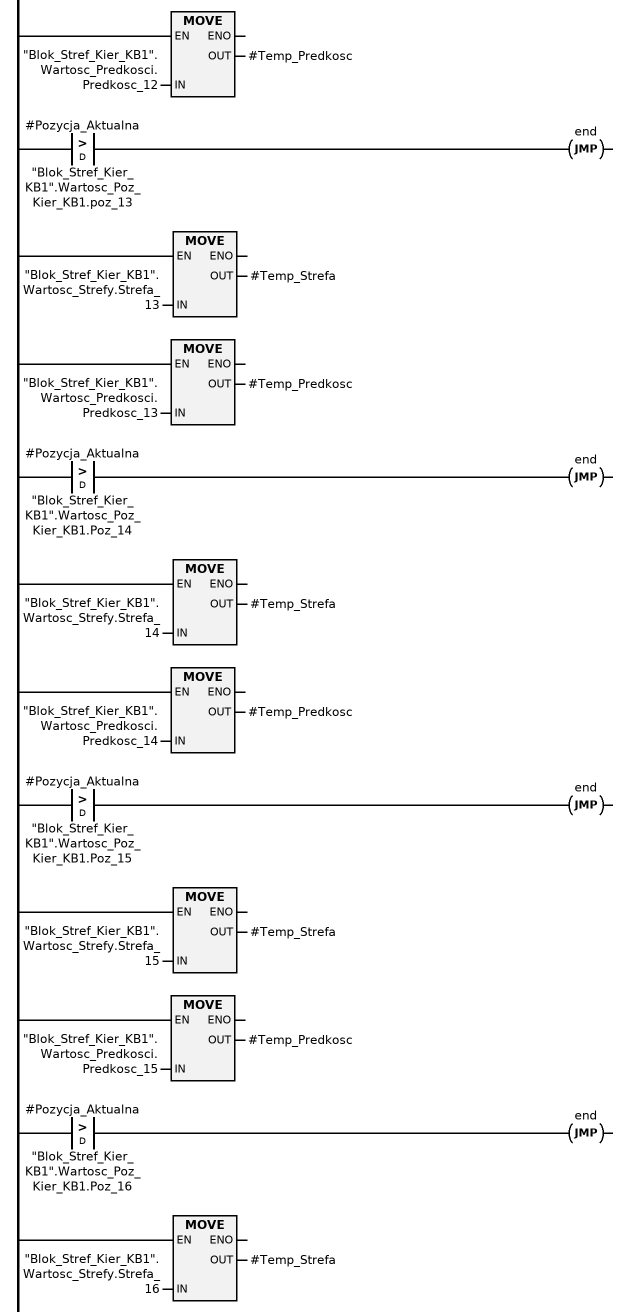
[picture p382: Przelaczanie_Stref_K_KB1 networks 3-3]
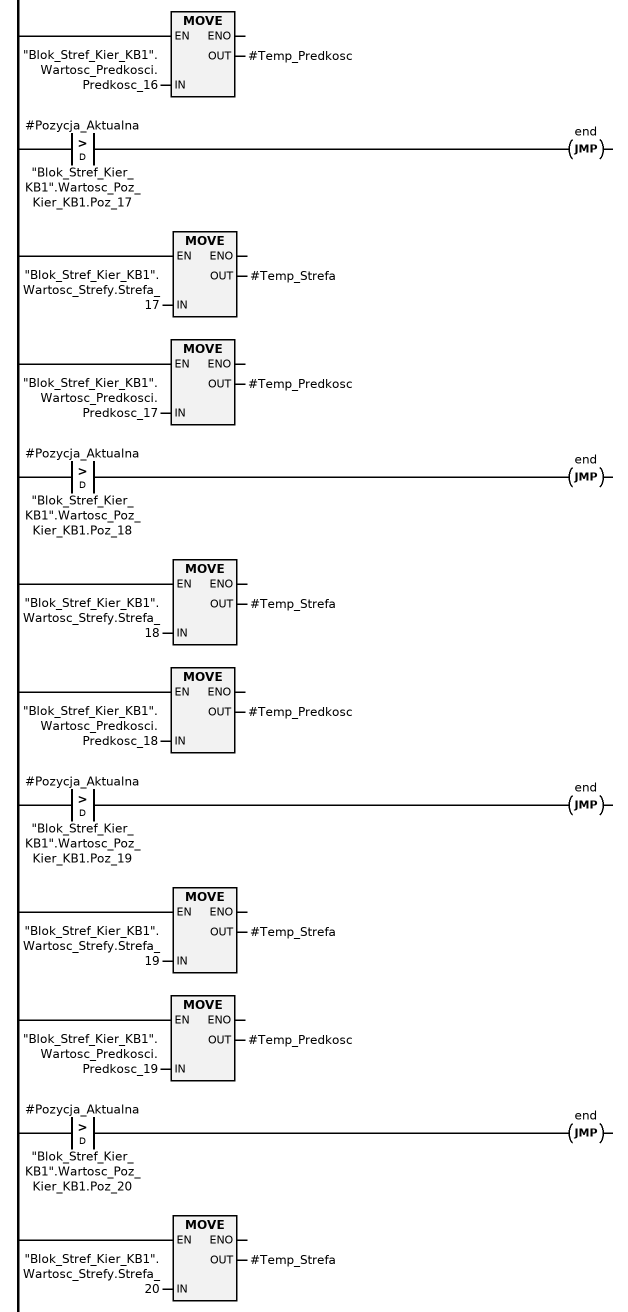
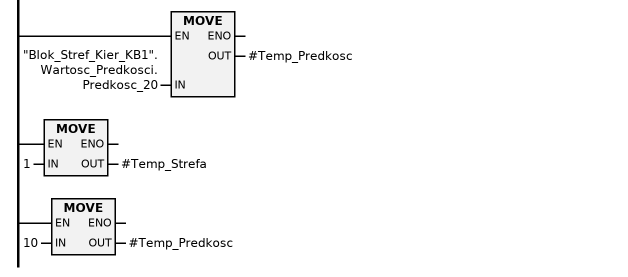
NETWORK
TITLE =
//Porowanie Pozycji z zadana strefa
//
//B1       
//
//5000               
//
//10000
//
//KB2
//                        /\
//                        |
//12000                 Wozek
//
//
//Gender
//15000
//*********Poz  0
      L     #Pozycja_Aktualna;	//np 350000
      L     "Blok_Stref_Kier_KB1".Wartosc_Poz_Kier_KB1.Poz_0;	//np40000 idzie dalej
      >D;
      JC    end;
      L     "Blok_Stref_Kier_KB1".Wartosc_Strefy.Strefa_0;
      T     #Temp_Strefa;
      L     "Blok_Stref_Kier_KB1".Wartosc_Predkosci.Predkosc_0;
      T     #Temp_Predkosc;
//*********Poz  1
      L     #Pozycja_Aktualna;	//30000
      L     "Blok_Stref_Kier_KB1".Wartosc_Poz_Kier_KB1.Poz_1;	//np.24000 tu zostaje
      >D;
      JC    end;
      L     "Blok_Stref_Kier_KB1".Wartosc_Strefy.Strefa_1;
      T     #Temp_Strefa;
      L     "Blok_Stref_Kier_KB1".Wartosc_Predkosci.Predkosc_1;
      T     #Temp_Predkosc;
//********Poz 2
      L     #Pozycja_Aktualna;	//20000
      L     "Blok_Stref_Kier_KB1".Wartosc_Poz_Kier_KB1.Poz_2;	//np22000
      >D;
      JC    end;
      L     "Blok_Stref_Kier_KB1".Wartosc_Strefy.Strefa_2;
      T     #Temp_Strefa;
      L     "Blok_Stref_Kier_KB1".Wartosc_Predkosci.Predkosc_2;
      T     #Temp_Predkosc;
//********Poz 3
      L     #Pozycja_Aktualna;
      L     "Blok_Stref_Kier_KB1".Wartosc_Poz_Kier_KB1.Poz_3;
      >D;
      JC    end;
      L     "Blok_Stref_Kier_KB1".Wartosc_Strefy.Strefa_3;
      T     #Temp_Strefa;
      L     "Blok_Stref_Kier_KB1".Wartosc_Predkosci.Predkosc_3;
      T     #Temp_Predkosc;
//********Poz 4
      L     #Pozycja_Aktualna;
      L     "Blok_Stref_Kier_KB1".Wartosc_Poz_Kier_KB1.Poz_4;
      >D;
      JC    end;
      L     "Blok_Stref_Kier_KB1".Wartosc_Strefy.Strefa_4;
      T     #Temp_Strefa;
      L     "Blok_Stref_Kier_KB1".Wartosc_Predkosci.Predkosc_4;
      T     #Temp_Predkosc;
//********Poz 5
      L     #Pozycja_Aktualna;
      L     "Blok_Stref_Kier_KB1".Wartosc_Poz_Kier_KB1.Poz_5;
      >D;
      JC    end;
      L     "Blok_Stref_Kier_KB1".Wartosc_Strefy.Strefa_5;
      T     #Temp_Strefa;
      L     "Blok_Stref_Kier_KB1".Wartosc_Predkosci.Predkosc_5;
      T     #Temp_Predkosc;
//********Poz 6
      L     #Pozycja_Aktualna;
      L     "Blok_Stref_Kier_KB1".Wartosc_Poz_Kier_KB1.Poz_6;
      >D;
      JC    end;
      L     "Blok_Stref_Kier_KB1".Wartosc_Strefy.Strefa_6;
      T     #Temp_Strefa;
      L     "Blok_Stref_Kier_KB1".Wartosc_Predkosci.Predkosc_6;
      T     #Temp_Predkosc;
//********Poz 7
      L     #Pozycja_Aktualna;
      L     "Blok_Stref_Kier_KB1".Wartosc_Poz_Kier_KB1.Poz_7;
      >D;
      JC    end;
      L     "Blok_Stref_Kier_KB1".Wartosc_Strefy.Strefa_7;
      T     #Temp_Strefa;
      L     "Blok_Stref_Kier_KB1".Wartosc_Predkosci.Predkosc_7;
      T     #Temp_Predkosc;
//********Poz 8
      L     #Pozycja_Aktualna;
      L     "Blok_Stref_Kier_KB1".Wartosc_Poz_Kier_KB1.Poz_8;
      >D;
      JC    end;
      L     "Blok_Stref_Kier_KB1".Wartosc_Strefy.Strefa_8;
      T     #Temp_Strefa;
      L     "Blok_Stref_Kier_KB1".Wartosc_Predkosci.Predkosc_8;
      T     #Temp_Predkosc;
//********Poz 9
      L     #Pozycja_Aktualna;
      L     "Blok_Stref_Kier_KB1".Wartosc_Poz_Kier_KB1.Poz_9;
      >D;
      JC    end;
      L     "Blok_Stref_Kier_KB1".Wartosc_Strefy.Strefa_9;
      T     #Temp_Strefa;
      L     "Blok_Stref_Kier_KB1".Wartosc_Predkosci.Predkosc_9;
      T     #Temp_Predkosc;
//********Poz 10
      L     #Pozycja_Aktualna;
      L     "Blok_Stref_Kier_KB1".Wartosc_Poz_Kier_KB1.Poz_10;
      >D;
      JC    end;
      L     "Blok_Stref_Kier_KB1".Wartosc_Strefy.Strefa_10;
      T     #Temp_Strefa;
      L     "Blok_Stref_Kier_KB1".Wartosc_Predkosci.Predkosc_10;
      T     #Temp_Predkosc;
//********Poz 11
      L     #Pozycja_Aktualna;
      L     "Blok_Stref_Kier_KB1".Wartosc_Poz_Kier_KB1.Poz_11;
      >D;
      JC    end;
      L     "Blok_Stref_Kier_KB1".Wartosc_Strefy.Strefa_11;
      T     #Temp_Strefa;
      L     "Blok_Stref_Kier_KB1".Wartosc_Predkosci.Predkosc_11;
      T     #Temp_Predkosc;
//********Poz 12
      L     #Pozycja_Aktualna;
      L     "Blok_Stref_Kier_KB1".Wartosc_Poz_Kier_KB1.Poz_12;
      >D;
      JC    end;
      L     "Blok_Stref_Kier_KB1".Wartosc_Strefy.Strefa_12;
      T     #Temp_Strefa;
      L     "Blok_Stref_Kier_KB1".Wartosc_Predkosci.Predkosc_12;
      T     #Temp_Predkosc;
//********Poz 13
      L     #Pozycja_Aktualna;
      L     "Blok_Stref_Kier_KB1".Wartosc_Poz_Kier_KB1.poz_13;
      >D;
      JC    end;
      L     "Blok_Stref_Kier_KB1".Wartosc_Strefy.Strefa_13;
      T     #Temp_Strefa;
      L     "Blok_Stref_Kier_KB1".Wartosc_Predkosci.Predkosc_13;
      T     #Temp_Predkosc;
//********Poz 14
      L     #Pozycja_Aktualna;
      L     "Blok_Stref_Kier_KB1".Wartosc_Poz_Kier_KB1.Poz_14;
      >D;
      JC    end;
      L     "Blok_Stref_Kier_KB1".Wartosc_Strefy.Strefa_14;
      T     #Temp_Strefa;
      L     "Blok_Stref_Kier_KB1".Wartosc_Predkosci.Predkosc_14;
      T     #Temp_Predkosc;
//********Poz 15
      L     #Pozycja_Aktualna;
      L     "Blok_Stref_Kier_KB1".Wartosc_Poz_Kier_KB1.Poz_15;
      >D;
      JC    end;
      L     "Blok_Stref_Kier_KB1".Wartosc_Strefy.Strefa_15;
      T     #Temp_Strefa;
      L     "Blok_Stref_Kier_KB1".Wartosc_Predkosci.Predkosc_15;
      T     #Temp_Predkosc;
//********Poz 16
      L     #Pozycja_Aktualna;
      L     "Blok_Stref_Kier_KB1".Wartosc_Poz_Kier_KB1.Poz_16;
      >D;
      JC    end;
      L     "Blok_Stref_Kier_KB1".Wartosc_Strefy.Strefa_16;
      T     #Temp_Strefa;
      L     "Blok_Stref_Kier_KB1".Wartosc_Predkosci.Predkosc_16;
      T     #Temp_Predkosc;
//********Poz 17
      L     #Pozycja_Aktualna;
      L     "Blok_Stref_Kier_KB1".Wartosc_Poz_Kier_KB1.Poz_17;
      >D;
      JC    end;
      L     "Blok_Stref_Kier_KB1".Wartosc_Strefy.Strefa_17;
      T     #Temp_Strefa;
      L     "Blok_Stref_Kier_KB1".Wartosc_Predkosci.Predkosc_17;
      T     #Temp_Predkosc;
//********Poz 18
      L     #Pozycja_Aktualna;
      L     "Blok_Stref_Kier_KB1".Wartosc_Poz_Kier_KB1.Poz_18;
      >D;
      JC    end;
      L     "Blok_Stref_Kier_KB1".Wartosc_Strefy.Strefa_18;
      T     #Temp_Strefa;
      L     "Blok_Stref_Kier_KB1".Wartosc_Predkosci.Predkosc_18;
      T     #Temp_Predkosc;
//********Poz 19
      L     #Pozycja_Aktualna;
      L     "Blok_Stref_Kier_KB1".Wartosc_Poz_Kier_KB1.Poz_19;
      >D;
      JC    end;
      L     "Blok_Stref_Kier_KB1".Wartosc_Strefy.Strefa_19;
      T     #Temp_Strefa;
      L     "Blok_Stref_Kier_KB1".Wartosc_Predkosci.Predkosc_19;
      T     #Temp_Predkosc;
//********Poz 20
      L     #Pozycja_Aktualna;
      L     "Blok_Stref_Kier_KB1".Wartosc_Poz_Kier_KB1.Poz_20;
      >D;
      JC    end;
      L     "Blok_Stref_Kier_KB1".Wartosc_Strefy.Strefa_20;
      T     #Temp_Strefa;
      L     "Blok_Stref_Kier_KB1".Wartosc_Predkosci.Predkosc_20;
      T     #Temp_Predkosc;
//Jezeli nic nie wyszlo wybierz strefe najwieksza
      L     1;
      T     #Temp_Strefa;
      L     10;
      T     #Temp_Predkosc;
end:  NOP   0;
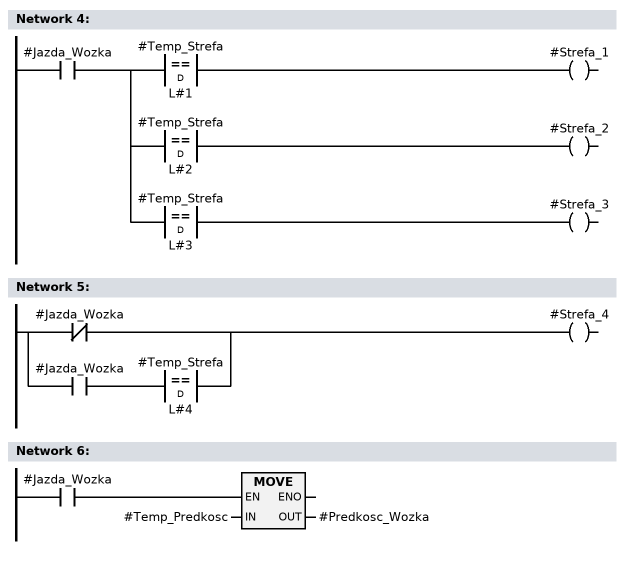
NETWORK
TITLE =
//Przypisanie predkosc. Strefa 1 to strefa podluzna.
//
      A     #Jazda_Wozka;
      =     L 8.0;
      A     L 8.0;
      A(;
      L     #Temp_Strefa;
      L     L#1;
      ==D;
      );
      =     #Strefa_1;
      A     L 8.0;
      A(;
      L     #Temp_Strefa;
      L     L#2;
      ==D;
      );
      =     #Strefa_2;
      A     L 8.0;
      A(;
      L     #Temp_Strefa;
      L     L#3;
      ==D;
      );
      =     #Strefa_3;
NETWORK
TITLE =
//Jezeli wozek stoi
      ON    #Jazda_Wozka;
      O;
      A     #Jazda_Wozka;
      A(;
      L     #Temp_Strefa;
      L     L#4;
      ==D;
      );
      =     #Strefa_4;
NETWORK
TITLE =
//Przyporzadkowanie predkosci
      A     #Jazda_Wozka;
      JNB   _001;
      L     #Temp_Predkosc;
      T     #Predkosc_Wozka;
_001: NOP   0;
END_FUNCTION

FUNCTION "Blok_Bedow" : VOID	// FC 119
//Funkcja obslugujaca bledy
VERSION : 0.1
BEGIN
NETWORK
TITLE =
//Ten network celowo jest wolny
//
NETWORK
TITLE =
END_FUNCTION

FUNCTION "Fal_Sew" : VOID	// FC 140
//Dieses Programmbeispiel zeigt nur die prinzipielle Vorgehensweise.
//Für fehlerhafte Programmfunktionen und deren Folgen
//kann weder eine juristische, noch irgendeine Haftung übernommen werden!
//
//Eingänge der FC:
//"DRIVE_IO_ADDRESS": Anfangsadresse des E/A-Bereichs => Hardwarekonfiguration
//"ENABLE_RAPID_STOP" = true: Freigabe; false: Schnellstopp
//"RESET": Fehler quittieren
//Die Betriebsart wird mit den Eingängen "Jog_plus_mode, Jog_minus_mode; 
//Ref_travel und Positioning_mode angewählt.
//"SETPOINT_POS": Positionssollwert (DINT) in Anwendereinheit.
//Die Anwendereinheit ist abhängig von der Inbetriebnahme der "Erweiterten 
//Buspositionierung"
//"SETPOINT_SPEED": Positioniergeschwindigkeit (INT) in rpm
//"START_RAMP": Beschleunigungsrampe (INT) in ms
//"STOP_RAMP": Verzögerungsrampe(INT) in ms
AUTHOR : SG-MEST
FAMILY : PROFIBUS
NAME : MDX_POS
VERSION : 1.1
VAR_INPUT
  DRIVE_IO_ADDRESS : INT ;
  ENABLE_RAPID_STOP : BOOL ;
  RESET : BOOL ;
  JOG_PLUS_MODE : BOOL ;
  JOG_MINUS_MODE : BOOL ;
  REF_TRAVEL_MODE : BOOL ;
  POSITIONING_MODE : BOOL ;
  SETPOINT_POS : DINT ;	//in mm
  SETPOINT_SPEED : INT ;	//Positioniergeschwindigkeit (INT) in rpm (1350rpm)
  START_RAMP : INT ;	//Beschleunigungsrampe (INT) in ms
  STOP_RAMP : INT ;	//Verzögerungsrampe(INT) in ms
END_VAR
VAR_OUTPUT
  COMMUNICATION_OK : BOOL ;	//SFC14/SFC15: Return Value = 0
  FAULT_OF_AXIS : BOOL ;
  WARNING_OF_AXIS : BOOL ;
  INVERTER_READY : BOOL ;
  REFERENCED : BOOL ;
  TARGET_POS_REACHED : BOOL ;
  AXIS_INTERLOCKED : BOOL ;	//die Modeanwahl ist unplausibel (kein Mode oder mehrere Modi angewählt)
  FAULT_NO : INT ;
  ACTUAL_POSITION : DINT ;
  ACTUAL_SPEED : INT ;
  ACTUAL_CURRENT : INT ;
END_VAR
VAR_TEMP
  PI : STRUCT
   Status : BYTE ;
   Motor_turning : BOOL ;
   Inverter_ready : BOOL ;
   referenced : BOOL ;
   Target_position_reached : BOOL ;
   Brake_released : BOOL ;
   Error : BOOL ;
   Limit_Switch_CW : BOOL ;
   Limit_switch_CCW : BOOL ;
   Actual_position : DINT ;
   Actual_speed : INT ;
   Active_current : INT ;
   Device_utilisation : INT ;
  END_STRUCT ;
  PO : STRUCT
   start : BOOL ;
   Jog_plus : BOOL ;
   Jog_minus : BOOL ;
   mode_low : BOOL ;
   mode_high : BOOL ;
   CTW_Bit_13 : BOOL ;
   CTW_Bit_14 : BOOL ;
   CTW_Bit_15 : BOOL ;
   Contr_inhibit : BOOL ;
   Rapid_stop : BOOL ;
   Stop : BOOL ;
   CTW_Bit_3 : BOOL ;
   CTW_Bit_4 : BOOL ;
   CTW_Bit_5 : BOOL ;
   Reset_fault : BOOL ;
   CTW_Bit_7 : BOOL ;
   Setpoint_position : DINT ;
   Setpoint_speed : INT ;
   Start_ramp : INT ;
   Stop_ramp : INT ;
  END_STRUCT ;
  Ref : BOOL ;
  Pos : BOOL ;
  Addr : WORD ;
  Returncode_SFC14 : INT ;
  Returncode_SFC15 : INT ;
END_VAR
BEGIN
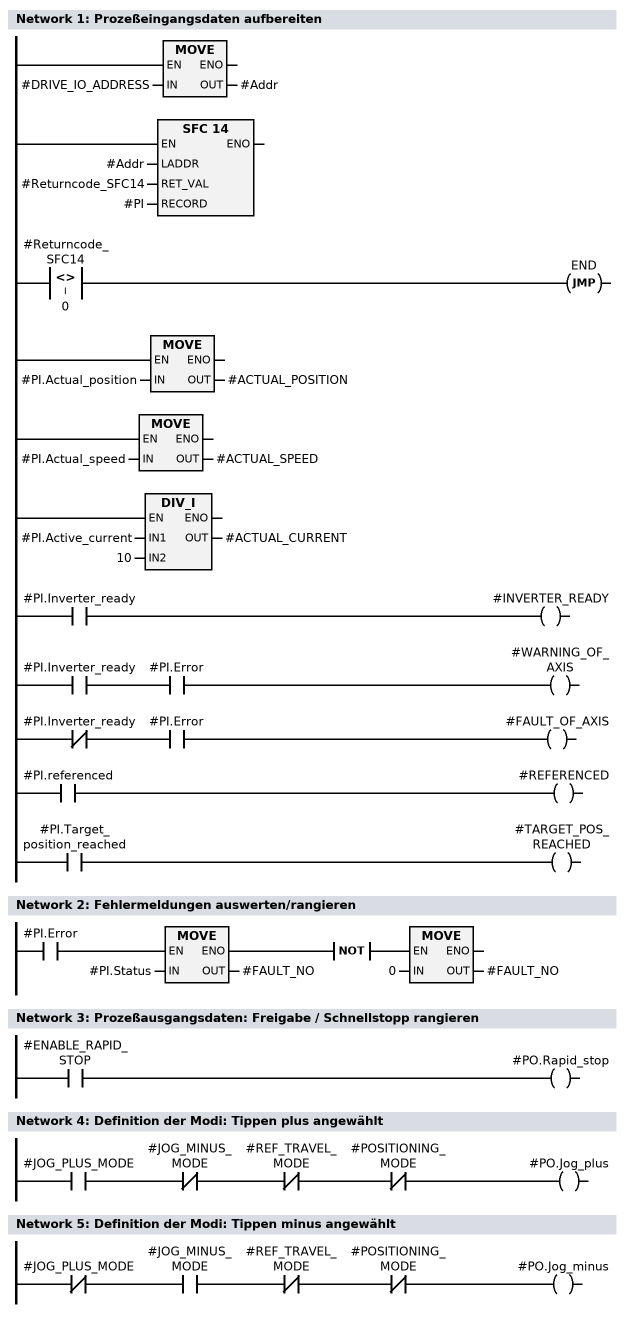
NETWORK
TITLE = Prozeßeingangsdaten aufbereiten
      L     #DRIVE_IO_ADDRESS;	//Adresse von "INT" nach "WORD" wandeln
      T     #Addr;
      CALL  SFC 14 (
           LADDR                    := #Addr,
           RET_VAL                  := #Returncode_SFC14,
           RECORD                   := #PI);	//konsistente Daten eines DP-Nomrslaves lesen / Peripherieadresse => Hardwarekonfig. / <> 0 => ein Fehler ist während der Bearbeitung aufgetreten / Zielbereich für die gelesenen Nutzdaten.
      L     #Returncode_SFC14;
      L     0;
      <>I;	//Tritt während der Abarbeitung der SFC ein Fehler auf,
      JC    END;	//so wird die Funktion verlassen => NW14
      L     #PI.Actual_position;	//Rangieren der Prozeßeingangsdaten
      T     #ACTUAL_POSITION;
      L     #PI.Actual_speed;
      T     #ACTUAL_SPEED;
      L     #PI.Active_current;
      L     10;
      /I;
      T     #ACTUAL_CURRENT;
      A     #PI.Inverter_ready;
      =     #INVERTER_READY;
      A     #PI.Inverter_ready;	//Eine Warnung ist aktiv, wenn der Umrichter noch betriebsbereit ist
      A     #PI.Error;	//und das Fehlerbit gesetzt ist.
      =     #WARNING_OF_AXIS;
      AN    #PI.Inverter_ready;	//Ein Fehler liegt vor, wenn der Umrichter nicht betriebsbereit ist
      A     #PI.Error;	//und das Fehlerbit gesetzt ist.
      =     #FAULT_OF_AXIS;
      A     #PI.referenced;
      =     #REFERENCED;
      A     #PI.Target_position_reached;
      =     #TARGET_POS_REACHED;
NETWORK
TITLE = Fehlermeldungen auswerten/rangieren
//Ist das Fehlerbit gesetzt, so wird die Fehlernummer ausgegeben.
//Liegt kein Fehler vor, so wird eine Null ausgegeben.
      A(;
      A     #PI.Error;
      JNB   _001;
      L     #PI.Status;
      T     #FAULT_NO;
      SET;
      SAVE;
      CLR;
_001: A     BR;
      );
      NOT;
      JNB   _002;
      L     0;
      T     #FAULT_NO;
_002: NOP   0;
NETWORK
TITLE = Prozeßausgangsdaten: Freigabe / Schnellstopp rangieren
      A     #ENABLE_RAPID_STOP;
      =     #PO.Rapid_stop;
NETWORK
TITLE = Definition der Modi: Tippen plus angewählt
      A     #JOG_PLUS_MODE;
      AN    #JOG_MINUS_MODE;
      AN    #REF_TRAVEL_MODE;
      AN    #POSITIONING_MODE;
      =     #PO.Jog_plus;
NETWORK
TITLE = Definition der Modi: Tippen minus angewählt
      AN    #JOG_PLUS_MODE;
      A     #JOG_MINUS_MODE;
      AN    #REF_TRAVEL_MODE;
      AN    #POSITIONING_MODE;
      =     #PO.Jog_minus;
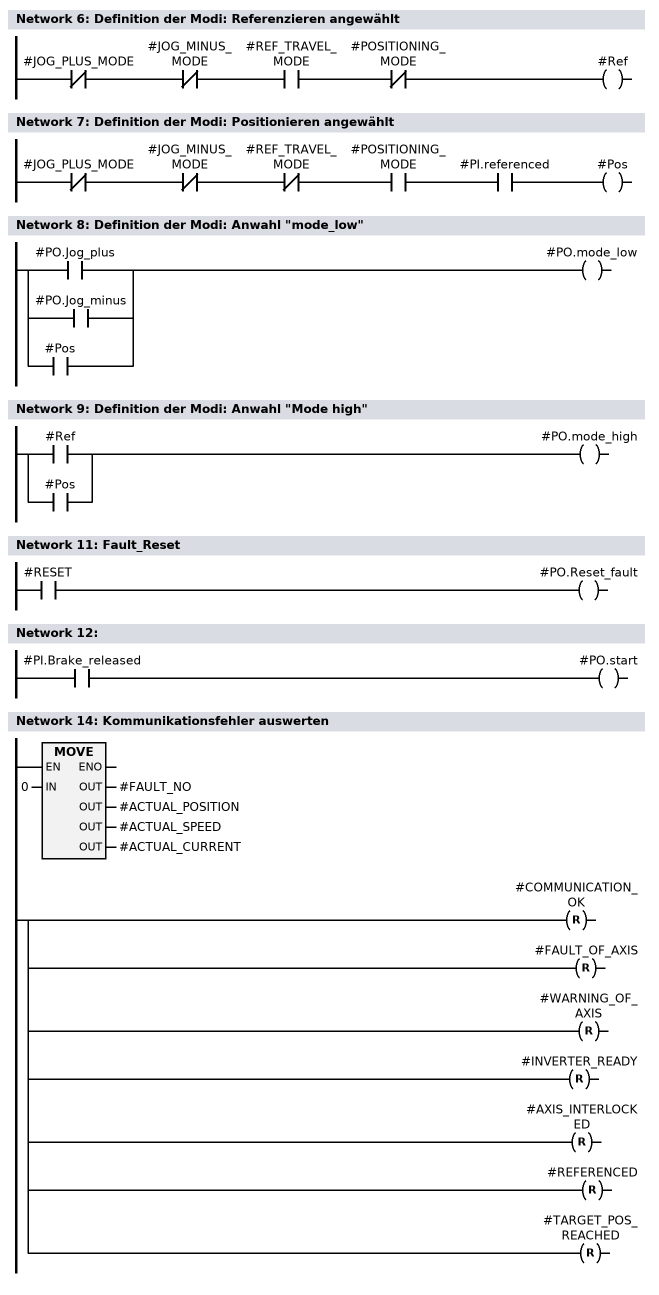
NETWORK
TITLE = Definition der Modi: Referenzieren angewählt
      AN    #JOG_PLUS_MODE;
      AN    #JOG_MINUS_MODE;
      A     #REF_TRAVEL_MODE;
      AN    #POSITIONING_MODE;
      =     #Ref;
NETWORK
TITLE = Definition der Modi: Positionieren angewählt
      AN    #JOG_PLUS_MODE;
      AN    #JOG_MINUS_MODE;
      AN    #REF_TRAVEL_MODE;
      A     #POSITIONING_MODE;
      A     #PI.referenced;
      =     #Pos;
NETWORK
TITLE = Definition der Modi: Anwahl "mode_low"
      O     #PO.Jog_plus;
      O     #PO.Jog_minus;
      O     #Pos;
      =     #PO.mode_low;
NETWORK
TITLE = Definition der Modi: Anwahl "Mode high"
      O     #Ref;
      O     #Pos;
      =     #PO.mode_high;
NETWORK
TITLE = Freigabe / Halt via Feldbus
      O     #PO.mode_low;
      O     #PO.mode_high;
      =     L 32.0;
      A     L 32.0;
      BLD   102;
      =     #PO.Stop;
      AN    L 32.0;
      =     #AXIS_INTERLOCKED;
NETWORK
TITLE = Fault_Reset
      A     #RESET;
      =     #PO.Reset_fault;
NETWORK
TITLE =
      A     #PI.Brake_released;
      =     #PO.start;
NETWORK
TITLE = Prozeßausgangsdaten: Sollwerte aufbereiten
      SET;
      R     #PO.Contr_inhibit;	//Rücksetzen aller nicht verwendeten Steuerwort-Bits
      R     #PO.CTW_Bit_3;
      R     #PO.CTW_Bit_4;
      R     #PO.CTW_Bit_5;
      R     #PO.CTW_Bit_13;
      R     #PO.CTW_Bit_14;
      R     #PO.CTW_Bit_15;
      L     #SETPOINT_POS;
      T     #PO.Setpoint_position;
      L     #SETPOINT_SPEED;
      T     #PO.Setpoint_speed;
      L     #START_RAMP;
      T     #PO.Start_ramp;
      L     #STOP_RAMP;
      T     #PO.Stop_ramp;
      CALL  SFC 15 (
           LADDR                    := #Addr,
           RECORD                   := #PO,
           RET_VAL                  := #Returncode_SFC15);	//Daten konsistent auf einen DP-Normslave schreiben / Peripherieadresse => Hardwarekonfig. / Quellbereich für die zu schreibenden Nutzdaten / <> 0 => ein Fehler istwährend der Bearbeitung aufgetreten
      L     #Returncode_SFC15;	//Tritt während der Abarbeitung des SFCs ein Fehler auf, 
      L     0;
      <>I;
      JC    END;	//so wird die Funktion verlassen. => NW14
      SET;
      =     #COMMUNICATION_OK;
      BEU;	//Ende der Funktion
NETWORK
TITLE = Kommunikationsfehler auswerten
//Ist die Abarbeitung der SFCs fehlerhaft, so werden alle Ausgänge der Funktion 
//abgelöscht
//
END:  L     0;
      T     #FAULT_NO;
      T     #ACTUAL_POSITION;
      T     #ACTUAL_SPEED;
      T     #ACTUAL_CURRENT;
      SET;
      R     #COMMUNICATION_OK;
      R     #FAULT_OF_AXIS;
      R     #WARNING_OF_AXIS;
      R     #INVERTER_READY;
      R     #AXIS_INTERLOCKED;
      R     #REFERENCED;
      R     #TARGET_POS_REACHED;
END_FUNCTION

FUNCTION "Predkosc_Fal" : VOID	// FC 141
//Kilkostopniowe ustalenie predkosci falownika. Funkcja zmniejsza predkosc o 
//wartosc procentowa. Na niewykorzystane wejscia daj wartosc 100
VERSION : 0.1
VAR_INPUT
  id_Wartosc_Predk : INT ;
  _1_Stopien : INT ;
  _2_Stopien : INT ;
  _3_Stopien : INT ;
  _4_Stopien : INT ;
  _5_Stopien : INT ;
  _6_Stopien : INT ;
END_VAR
VAR_OUTPUT
  ow_Predkosc_Wyjsciowa : INT ;
END_VAR
VAR_TEMP
  T_1_Stopien : REAL ;
  T_2_Stopien : REAL ;
  T_3_Stopien : REAL ;
  T_4_Stopien : REAL ;
  T_5_Stopien : REAL ;
  T_6_Stopien : REAL ;
  T_Predkosc : REAL ;
  T_Help_Real : REAL ;
END_VAR
BEGIN
NETWORK
TITLE =
//Ten network celowo jest wolny
NETWORK
TITLE =
//Przeskalowanie stopnia na real
//Stopien 1 
      L     #_1_Stopien;
      ITD;
      DTR;
      L     1.000000e+02;
      /R;
      T     #T_1_Stopien;
//Stopien 2
      L     #_2_Stopien;
      ITD;
      DTR;
      L     1.000000e+02;
      /R;
      T     #T_2_Stopien;
//Stopien 3 
      L     #_3_Stopien;
      ITD;
      DTR;
      L     1.000000e+02;
      /R;
      T     #T_3_Stopien;
//Stopien 4 
      L     #_4_Stopien;
      ITD;
      DTR;
      L     1.000000e+02;
      /R;
      T     #T_4_Stopien;
//Stopien 5 
      L     #_5_Stopien;
      ITD;
      DTR;
      L     1.000000e+02;
      /R;
      T     #T_5_Stopien;
//Stopien 6 
      L     #_6_Stopien;
      ITD;
      DTR;
      L     1.000000e+02;
      /R;
      T     #T_6_Stopien;
//konwersja predkosci
      L     #id_Wartosc_Predk;
      ITD;
      DTR;
      T     #T_Predkosc;
NETWORK
TITLE =
//--1 stopien
      L     #T_Predkosc;
      L     #T_1_Stopien;
      *R;
      T     #T_Help_Real;
//--2
      L     #T_Help_Real;
      L     #T_2_Stopien;
      *R;
      T     #T_Help_Real;
//--3
      L     #T_Help_Real;
      L     #T_3_Stopien;
      *R;
      T     #T_Help_Real;
//--4
      L     #T_Help_Real;
      L     #T_4_Stopien;
      *R;
      T     #T_Help_Real;
//--5
      L     #T_Help_Real;
      L     #T_5_Stopien;
      *R;
      T     #T_Help_Real;
//--6
      L     #T_Help_Real;
      L     #T_6_Stopien;
      *R;
      T     #T_Help_Real;
      L     #T_Help_Real;
      RND;
      T     #ow_Predkosc_Wyjsciowa;
END_FUNCTION

FUNCTION "Funkcja_Zegara" : VOID	// FC 150
AUTHOR : Kng
NAME : HELP_FC
VERSION : 0.1
VAR_INPUT
  Timer_NR : TIMER ;
  Czas : S5TIME ;
END_VAR
VAR_IN_OUT
  Wyjscie : BOOL ;
END_VAR
BEGIN
NETWORK
TITLE =
      A     #Timer_NR;
      SAVE;
      NOT;
      L     #Czas;
      SD    #Timer_NR;
      X     BR;
      X     #Wyjscie;
      =     #Wyjscie;
END_FUNCTION

FUNCTION "COM_Odbieranie" : VOID	// FC 200
VERSION : 0.1
BEGIN
NETWORK
TITLE =
//Ten Network celowo jest wolny
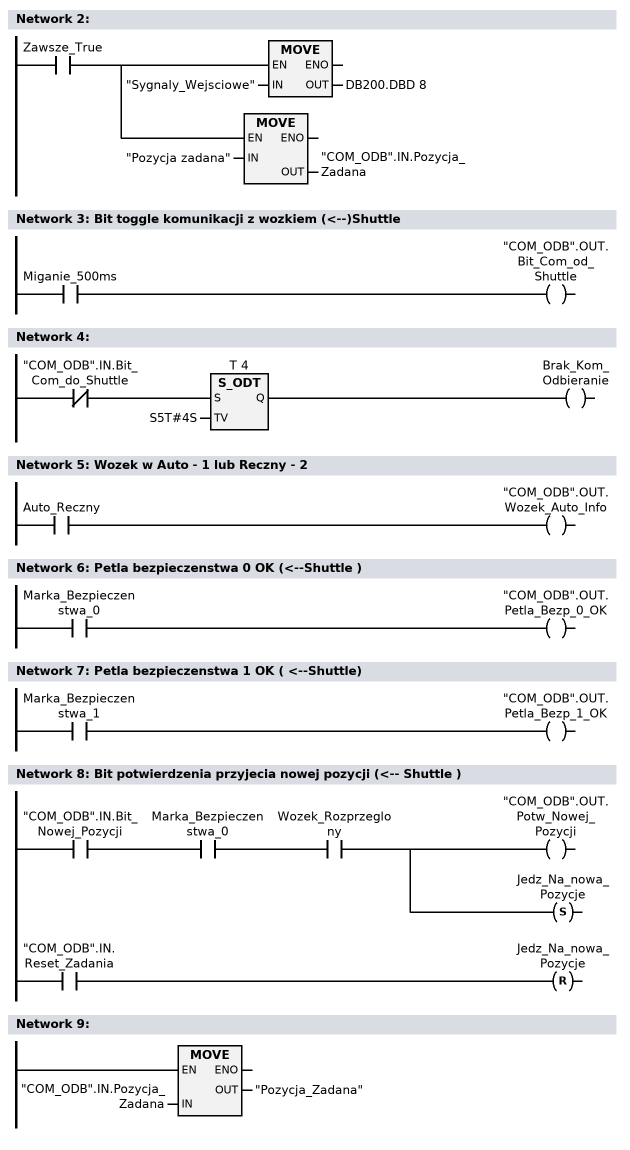
NETWORK
TITLE =
//Przepisywanie danych input 38 i 42
      A     "Zawsze_True";
      =     L 0.0;
      A     L 0.0;
      JNB   _001;
      L     "Sygnaly_Wejsciowe";
      T     DB200.DBD 8;
_001: NOP   0;
      A     L 0.0;
      JNB   _002;
      L     "Pozycja zadana";
      T     "COM_ODB".IN.Pozycja_Zadana;
_002: NOP   0;
NETWORK
TITLE = Bit toggle komunikacji z wozkiem (<--)Shuttle 
//Sprawdzenie komunikacji
      A     "Miganie_500ms";
      =     "COM_ODB".OUT.Bit_Com_od_Shuttle;
NETWORK
TITLE =
//sprawdzenie czy jest komunikacja
      AN    "COM_ODB".IN.Bit_Com_do_Shuttle;
      L     S5T#4S;
      SD    T 4;
      NOP   0;
      NOP   0;
      NOP   0;
      A     T 4;
      =     "Brak_Kom_Odbieranie";
NETWORK
TITLE = Wozek w Auto - 1 lub Reczny - 2
//Sprawdzenie czy wozek jest w trybie auto
      A     "Auto_Reczny";
      =     "COM_ODB".OUT.Wozek_Auto_Info;
NETWORK
TITLE = Petla bezpieczenstwa 0 OK (<--Shuttle )
//Przekazanie informacji o bezpieczenstwie
//
      A     "Marka_Bezpieczenstwa_0";
      =     "COM_ODB".OUT.Petla_Bezp_0_OK;
NETWORK
TITLE = Petla bezpieczenstwa 1 OK ( <--Shuttle)
//Petla 1 ok
      A     "Marka_Bezpieczenstwa_1";
      =     "COM_ODB".OUT.Petla_Bezp_1_OK;
NETWORK
TITLE = Bit potwierdzenia przyjecia nowej pozycji (<-- Shuttle )
//Odebranie nowego zadania
      A     "COM_ODB".IN.Bit_Nowej_Pozycji;
      A     "Marka_Bezpieczenstwa_0";
      A     "Wozek_Rozprzeglony";
      =     L 0.0;
      A     L 0.0;
      BLD   102;
      =     "COM_ODB".OUT.Potw_Nowej_Pozycji;
      A     L 0.0;
      S     "Jedz_Na_nowa_Pozycje";
      A     "COM_ODB".IN.Reset_Zadania;
      R     "Jedz_Na_nowa_Pozycje";
      NOP   0;
NETWORK
TITLE =
//Przepisanie pozycji zadanej
      L     "COM_ODB".IN.Pozycja_Zadana;
      T     "Pozycja_Zadana";
      NOP   0;
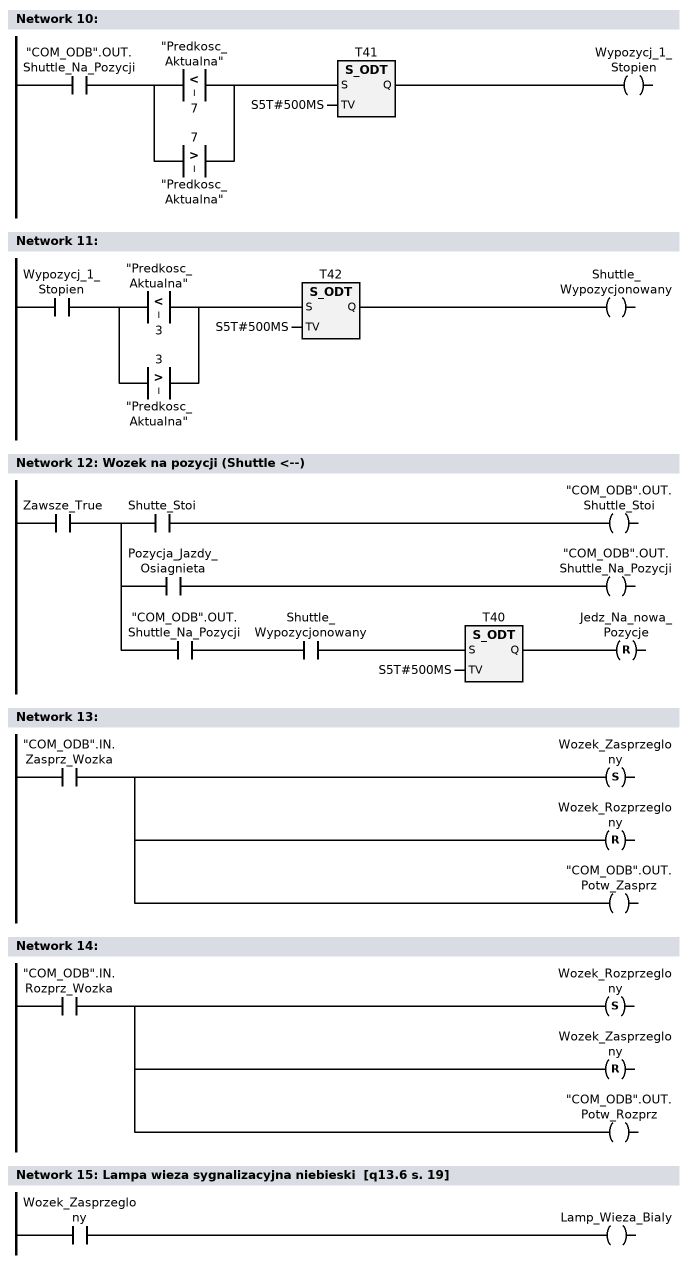
NETWORK
TITLE =
      A     "COM_ODB".OUT.Shuttle_Na_Pozycji;
      A(;
      O(;
      L     "Predkosc_Aktualna";
      L     7;
      <I;
      );
      O(;
      L     7;
      L     "Predkosc_Aktualna";
      >I;
      );
      );
      L     S5T#500MS;
      SD    "T41";
      NOP   0;
      NOP   0;
      NOP   0;
      A     "T41";
      =     "Wypozycj_1_Stopien";
NETWORK
TITLE =
      A     "Wypozycj_1_Stopien";
      A(;
      O(;
      L     "Predkosc_Aktualna";
      L     3;
      <I;
      );
      O(;
      L     3;
      L     "Predkosc_Aktualna";
      >I;
      );
      );
      L     S5T#500MS;
      SD    "T42";
      NOP   0;
      NOP   0;
      NOP   0;
      A     "T42";
      =     "Shuttle_Wypozycjonowany";
NETWORK
TITLE = Wozek na pozycji (Shuttle <--)
//Wozek nie jedzie
      A     "Zawsze_True";
      =     L 0.0;
      A     L 0.0;
      A     "Shutte_Stoi";
      =     "COM_ODB".OUT.Shuttle_Stoi;
      A     L 0.0;
      A     "Pozycja_Jazdy_Osiagnieta";
      =     "COM_ODB".OUT.Shuttle_Na_Pozycji;
      A     L 0.0;
      A     "COM_ODB".OUT.Shuttle_Na_Pozycji;
      A     "Shuttle_Wypozycjonowany";
      L     S5T#500MS;
      SD    "T40";
      NOP   0;
      NOP   0;
      NOP   0;
      A     "T40";
      R     "Jedz_Na_nowa_Pozycje";
NETWORK
TITLE =
//Zasprzeglenie wozka
      A     "COM_ODB".IN.Zasprz_Wozka;
      S     "Wozek_Zasprzeglony";
      R     "Wozek_Rozprzeglony";
      =     "COM_ODB".OUT.Potw_Zasprz;
NETWORK
TITLE =
//Rozsprzegniecie wozka
//
      A     "COM_ODB".IN.Rozprz_Wozka;
      S     "Wozek_Rozprzeglony";
      R     "Wozek_Zasprzeglony";
      =     "COM_ODB".OUT.Potw_Rozprz;
NETWORK
TITLE = Lampa wieza sygnalizacyjna niebieski  [q13.6 s. 19]
      A     "Wozek_Zasprzeglony";
      =     "Lamp_Wieza_Bialy";
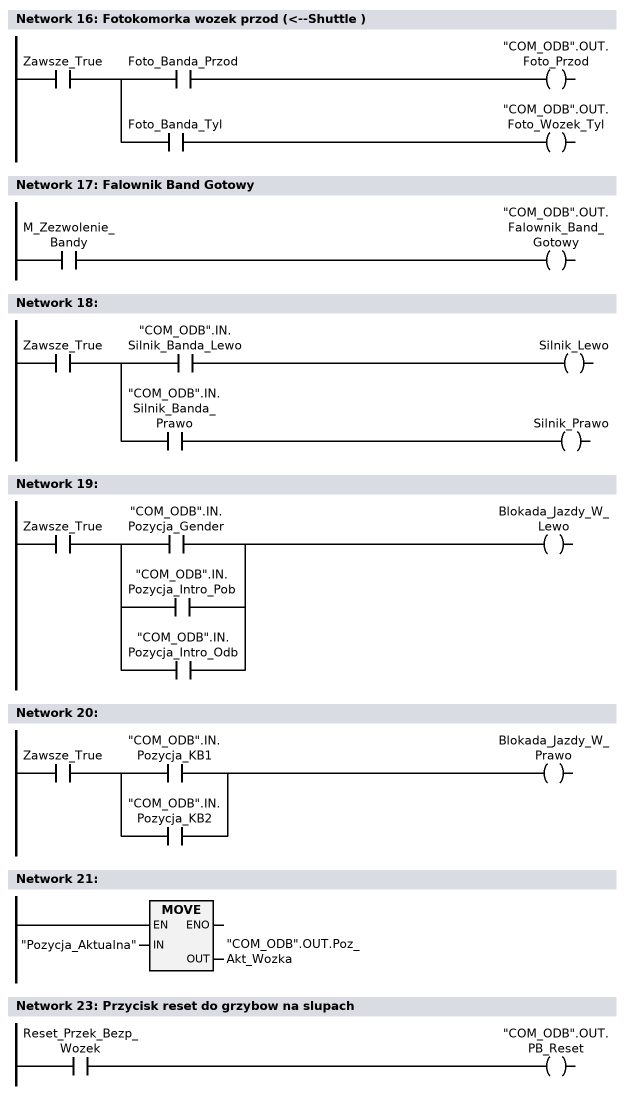
NETWORK
TITLE = Fotokomorka wozek przod (<--Shuttle )
//Przepisanie Fotokomorek
      A     "Zawsze_True";
      =     L 0.0;
      A     L 0.0;
      A     "Foto_Banda_Przod";
      =     "COM_ODB".OUT.Foto_Przod;
      A     L 0.0;
      A     "Foto_Banda_Tyl";
      =     "COM_ODB".OUT.Foto_Wozek_Tyl;
NETWORK
TITLE = Falownik Band Gotowy
      A     "M_Zezwolenie_Bandy";
      =     "COM_ODB".OUT.Falownik_Band_Gotowy;
NETWORK
TITLE =
//Jazda Silnikow
      A     "Zawsze_True";
      =     L 0.0;
      A     L 0.0;
      A     "COM_ODB".IN.Silnik_Banda_Lewo;
      =     "Silnik_Lewo";
      A     L 0.0;
      A     "COM_ODB".IN.Silnik_Banda_Prawo;
      =     "Silnik_Prawo";
NETWORK
TITLE =
//Informacja o blokadach jazdy. Sa one wlaczone jak za dlugo kreca rolki.
//Blokada w lewo.
      A     "Zawsze_True";
      A(;
      O     "COM_ODB".IN.Pozycja_Gender;
      O     "COM_ODB".IN.Pozycja_Intro_Pob;
      O     "COM_ODB".IN.Pozycja_Intro_Odb;
      );
      =     "Blokada_Jazdy_W_Lewo";
NETWORK
TITLE =
//Informacja o blokadach jazdy. Sa one wlaczone jak za dlugo kreca rolki.
//Blokada w prawo.
      A     "Zawsze_True";
      A(;
      O     "COM_ODB".IN.Pozycja_KB1;
      O     "COM_ODB".IN.Pozycja_KB2;
      );
      =     "Blokada_Jazdy_W_Prawo";
NETWORK
TITLE =
//Pozycja wozka aktualna
      L     "Pozycja_Aktualna";
      T     "COM_ODB".OUT.Poz_Akt_Wozka;
      NOP   0;
NETWORK
TITLE =
//Przepisanie wyjsc 
NETWORK
TITLE = Przycisk reset do grzybow na slupach
//Przyckisk reset
      A     "Reset_Przek_Bezp_Wozek";
      =     "COM_ODB".OUT.PB_Reset;
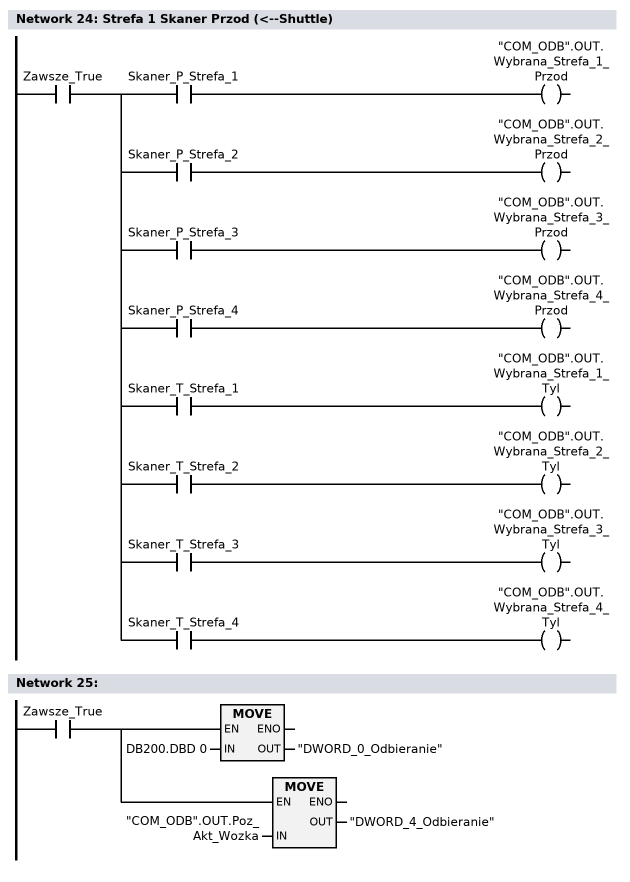
NETWORK
TITLE = Strefa 1 Skaner Przod (<--Shuttle)
//informacja o przelaczonych skanerach
      A     "Zawsze_True";
      =     L 0.0;
      A     L 0.0;
      A     "Skaner_P_Strefa_1";
      =     "COM_ODB".OUT.Wybrana_Strefa_1_Przod;
      A     L 0.0;
      A     "Skaner_P_Strefa_2";
      =     "COM_ODB".OUT.Wybrana_Strefa_2_Przod;
      A     L 0.0;
      A     "Skaner_P_Strefa_3";
      =     "COM_ODB".OUT.Wybrana_Strefa_3_Przod;
      A     L 0.0;
      A     "Skaner_P_Strefa_4";
      =     "COM_ODB".OUT.Wybrana_Strefa_4_Przod;
      A     L 0.0;
      A     "Skaner_T_Strefa_1";
      =     "COM_ODB".OUT.Wybrana_Strefa_1_Tyl;
      A     L 0.0;
      A     "Skaner_T_Strefa_2";
      =     "COM_ODB".OUT.Wybrana_Strefa_2_Tyl;
      A     L 0.0;
      A     "Skaner_T_Strefa_3";
      =     "COM_ODB".OUT.Wybrana_Strefa_3_Tyl;
      A     L 0.0;
      A     "Skaner_T_Strefa_4";
      =     "COM_ODB".OUT.Wybrana_Strefa_4_Tyl;
NETWORK
TITLE =
//Przypisanie wartosci wyjsciowych
      A     "Zawsze_True";
      =     L 0.0;
      A     L 0.0;
      JNB   _003;
      L     DB200.DBD 0;
      T     "DWORD_0_Odbieranie";
_003: NOP   0;
      A     L 0.0;
      JNB   _004;
      L     "COM_ODB".OUT.Poz_Akt_Wozka;
      T     "DWORD_4_Odbieranie";
_004: NOP   0;
NETWORK
TITLE =
      BEU;
NETWORK
TITLE =
END_FUNCTION

FUNCTION "COM_Pakiety" : VOID	// FC 201
VERSION : 0.1
BEGIN
NETWORK
TITLE =
//Ten Network celowo jest wolny
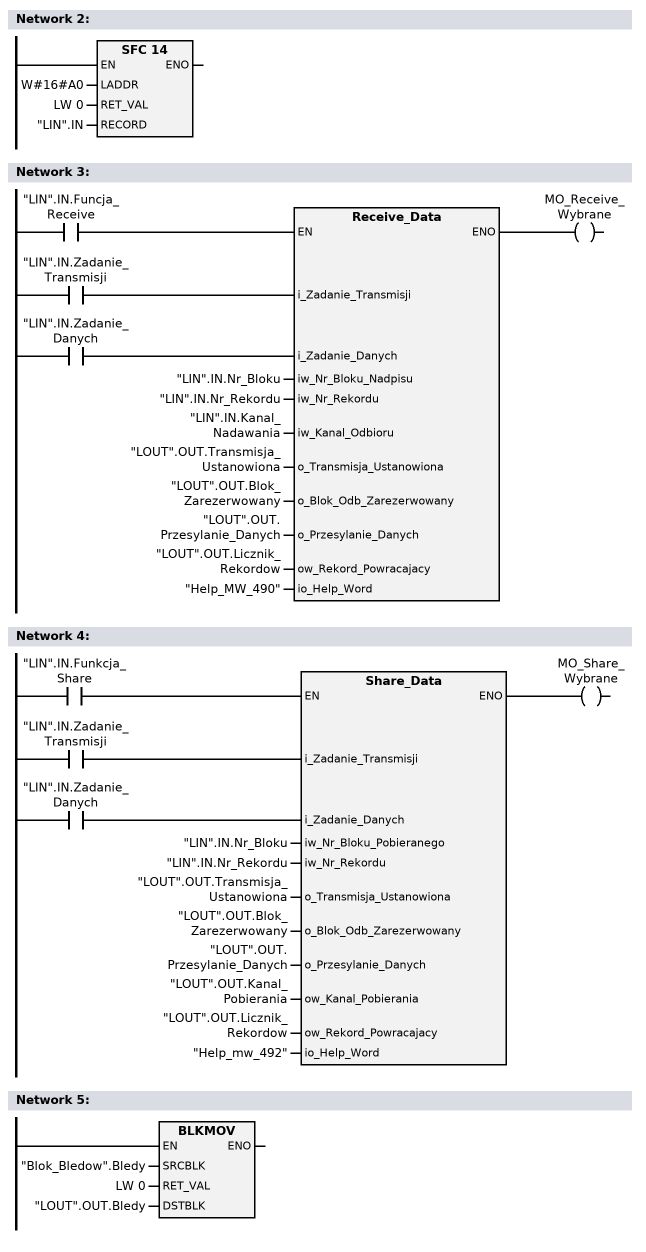
NETWORK
TITLE =
//Pobierz dane z mastera
//
//
      CALL  SFC 14 (
           LADDR                    := W#16#A0,
           RET_VAL                  := LW 0,
           RECORD                   := "LIN".IN);
      NOP   0;
NETWORK
TITLE =
//Odbieranie danych wysylanych z mastera
      A     "LIN".IN.Zadanie_Transmisji;
      =     L 2.0;
      BLD   103;
      A     "LIN".IN.Zadanie_Danych;
      =     L 2.1;
      BLD   103;
      A     "LIN".IN.Funcja_Receive;
      JNB   _001;
      CALL  "Receive_Data" (
           i_Zadanie_Transmisji     := L 2.0,
           i_Zadanie_Danych         := L 2.1,
           iw_Nr_Bloku_Nadpisu      := "LIN".IN.Nr_Bloku,
           iw_Nr_Rekordu            := "LIN".IN.Nr_Rekordu,
           iw_Kanal_Odbioru         := "LIN".IN.Kanal_Nadawania,
           o_Transmisja_Ustanowiona := "LOUT".OUT.Transmisja_Ustanowiona,
           o_Blok_Odb_Zarezerwowany := "LOUT".OUT.Blok_Zarezerwowany,
           o_Przesylanie_Danych     := "LOUT".OUT.Przesylanie_Danych,
           ow_Rekord_Powracajacy    := "LOUT".OUT.Licznik_Rekordow,
           io_Help_Word             := "Help_MW_490");
_001: A     BR;
      =     "MO_Receive_Wybrane";
NETWORK
TITLE =
//Odczyt danych
      A     "LIN".IN.Zadanie_Transmisji;
      =     L 2.0;
      BLD   103;
      A     "LIN".IN.Zadanie_Danych;
      =     L 2.1;
      BLD   103;
      A     "LIN".IN.Funkcja_Share;
      JNB   _002;
      CALL  "Share_Data" (
           i_Zadanie_Transmisji     := L 2.0,
           i_Zadanie_Danych         := L 2.1,
           iw_Nr_Bloku_Pobieranego  := "LIN".IN.Nr_Bloku,
           iw_Nr_Rekordu            := "LIN".IN.Nr_Rekordu,
           o_Transmisja_Ustanowiona := "LOUT".OUT.Transmisja_Ustanowiona,
           o_Blok_Odb_Zarezerwowany := "LOUT".OUT.Blok_Zarezerwowany,
           o_Przesylanie_Danych     := "LOUT".OUT.Przesylanie_Danych,
           ow_Kanal_Pobierania      := "LOUT".OUT.Kanal_Pobierania,
           ow_Rekord_Powracajacy    := "LOUT".OUT.Licznik_Rekordow,
           io_Help_Word             := "Help_mw_492");
_002: A     BR;
      =     "MO_Share_Wybrane";
NETWORK
TITLE =
//Przeniesienie bledow do czesci pakietowej
      CALL  "BLKMOV" (
           SRCBLK                   := "Blok_Bledow".Bledy,
           RET_VAL                  := LW 0,
           DSTBLK                   := "LOUT".OUT.Bledy);
      NOP   0;
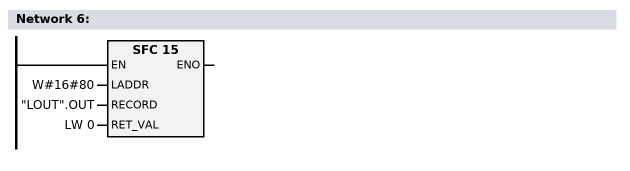
NETWORK
TITLE =
//Pobierz dane z mastera
//
//
      CALL  SFC 15 (
           LADDR                    := W#16#80,
           RECORD                   := "LOUT".OUT,
           RET_VAL                  := LW 0);
      NOP   0;
NETWORK
TITLE =
END_FUNCTION

FUNCTION "Receive_Data" : VOID	// FC 701
//Funkcja Share_Data udostepnia dane funkcji Read_Data. Sluzy do odczytu 
//parametrow z oddalonego urzadzenia przez waski kilku-bajtowy kanal 
//komunikacyjny.
//Poszczegolne kroki w wysylaniu i odbieraniu
//
//i_zadanie_transmisji     --> o_transmisja_ustanowiona
//iw_Nr_Bloku_Pobieranego  --> o_Blok_Pobierany_Zarezerwowany
//i_zadanie_danych         --> o_przesylanie_danych
//                         --> o_koniec_przesylania
//
//Po kazdej przeslanej danej musi dosjsc do inwersji bitu toggle
AUTHOR : Kng
NAME : COM
VERSION : 0.1
VAR_INPUT
  i_Zadanie_Transmisji : BOOL ;	//Ustanowienie transmisji
  i_Zadanie_Danych : BOOL ;	//Zadanie wyslania indeksu danych
  iw_Nr_Bloku_Nadpisu : INT ;
  iw_Nr_Rekordu : INT ;
  iw_Kanal_Odbioru : INT ;
END_VAR
VAR_OUTPUT
  o_Transmisja_Ustanowiona : BOOL ;	//Odpowiedz na zadanie transmisji
  o_Blok_Odb_Zarezerwowany : BOOL ;	//Potwierdzenie rezerwacji bloku
  o_Przesylanie_Danych : BOOL ;	//Przesylanie w toku
  ow_Rekord_Powracajacy : INT ;
END_VAR
VAR_IN_OUT
  io_Help_Word : WORD ;
END_VAR
VAR_TEMP
  Temp_Bool_1 : BOOL ;
  Temp_Byte : BYTE ;
  Help_Word_2 : WORD ;
  L_NR_Bloku_Danych : WORD ;
  L_Liczba_Rekordow : INT ;
  L_DW_Licznik_Rekordow : DWORD ;
END_VAR
BEGIN
NETWORK
TITLE =
//Ten Network celowo jest wolny
NETWORK
TITLE =
//Pobranie zmiennych pomocniczych
      L     #io_Help_Word;
      T     LW 0;
NETWORK
TITLE =
//Rzadanie transmisji
//
      A     #i_Zadanie_Transmisji;
      =     #o_Transmisja_Ustanowiona;
NETWORK
TITLE =
//Reset licznika rekordow
      A     #i_Zadanie_Transmisji;
      AN    #i_Zadanie_Danych;
      JCN   et_1;
      L     0;
      T     #ow_Rekord_Powracajacy;
et_1: NOP   0;
NETWORK
TITLE =
//Pobierz nazwe bloku kopiowanego
// sprawdzenie czy blok rozny od 0
      L     #iw_Nr_Bloku_Nadpisu;
      T     #L_NR_Bloku_Danych;
      L     0;
      <>I;
      =     #o_Blok_Odb_Zarezerwowany;
      A     #i_Zadanie_Transmisji;
      A     #i_Zadanie_Danych;
      =     #o_Przesylanie_Danych;
      AN    #o_Blok_Odb_Zarezerwowany;
      JC    end;
//Blok pobierany
      OPN   DB [#L_NR_Bloku_Danych];	// Otwarcie db
NETWORK
TITLE =
//Przeslanie Pierwszego podwojenego slowa w celu nawiazania komunikacji
// zamiania na double 
      L     #iw_Nr_Rekordu;
      L     2;
      *I;
      ITD;
      SLD   3;
      T     #L_DW_Licznik_Rekordow;
//Transmisja
      A     #o_Przesylanie_Danych;
      JCN   et_4;
      L     #iw_Kanal_Odbioru;
      T     DBW [#L_DW_Licznik_Rekordow];
      L     #iw_Nr_Rekordu;
      T     #ow_Rekord_Powracajacy;
et_4: NOP   0;
end:  NOP   0;
NETWORK
TITLE =
//Zapis bitow przejsciowych
      L     LW 0;
      T     #io_Help_Word;
      BEU;
END_FUNCTION

FUNCTION "Share_Data" : VOID	// FC 703
//Funkcja Share_Data udostepnia dane funkcji Read_Data. Sluzy do odczytu 
//parametrow z oddalonego urzadzenia przez waski kilku-bajtowy kanal 
//komunikacyjny.
//Poszczegolne kroki w wysylaniu i odbieraniu
//
//i_zadanie_transmisji     --> o_transmisja_ustanowiona
//iw_Nr_Bloku_Pobieranego  --> o_Blok_Pobierany_Zarezerwowany
//i_zadanie_danych         --> o_przesylanie_danych
//                         --> o_koniec_przesylania
//
//Po kazdej przeslanej danej musi dosjsc do inwersji bitu toggle
AUTHOR : Kng
NAME : COM
VERSION : 0.1
VAR_INPUT
  i_Zadanie_Transmisji : BOOL ;	//Ustanowienie transmisji
  i_Zadanie_Danych : BOOL ;	//Zadanie wyslania indeksu danych
  iw_Nr_Bloku_Pobieranego : INT ;
  iw_Nr_Rekordu : INT ;
END_VAR
VAR_OUTPUT
  o_Transmisja_Ustanowiona : BOOL ;	//Odpowiedz na zadanie transmisji
  o_Blok_Odb_Zarezerwowany : BOOL ;	//Potwierdzenie rezerwacji bloku
  o_Przesylanie_Danych : BOOL ;	//Przesylanie w toku
  ow_Kanal_Pobierania : INT ;	//Dane ktore sa udostepniane
  ow_Rekord_Powracajacy : INT ;
END_VAR
VAR_IN_OUT
  io_Help_Word : WORD ;
END_VAR
VAR_TEMP
  Temp_Bool_1 : BOOL ;
  Temp_Byte : BYTE ;
  Help_Word_2 : WORD ;
  L_NR_Bloku_Danych : WORD ;
  L_Liczba_Rekordow : INT ;
  L_DW_Licznik_Rekordow : DWORD ;
END_VAR
BEGIN
NETWORK
TITLE =
//Ten Network celowo jest wolny
NETWORK
TITLE =
//Pobranie zmiennych pomocniczych
      L     #io_Help_Word;
      T     LW 0;
NETWORK
TITLE =
//Rzadanie transmisji
//
      A     #i_Zadanie_Transmisji;
      =     #o_Transmisja_Ustanowiona;
      L     0;
      T     #ow_Rekord_Powracajacy;
NETWORK
TITLE =
//Reset licznika rekordow
      A     #i_Zadanie_Transmisji;
      AN    #i_Zadanie_Danych;
      JCN   et_1;
      L     0;
      T     #ow_Rekord_Powracajacy;
et_1: NOP   0;
NETWORK
TITLE =
//Pobierz nazwe bloku kopiowanego
// sprawdzenie czy blok rozny od 0
      L     #iw_Nr_Bloku_Pobieranego;
      T     #L_NR_Bloku_Danych;
      L     0;
      <>I;
      =     #o_Blok_Odb_Zarezerwowany;
      A     #i_Zadanie_Transmisji;
      A     #i_Zadanie_Danych;
      =     #o_Przesylanie_Danych;
      AN    #o_Blok_Odb_Zarezerwowany;
      JC    end;
//Blok pobierany
      OPN   DB [#L_NR_Bloku_Danych];	// Otwarcie db
NETWORK
TITLE =
//Przeslanie Pierwszego podwojenego slowa w celu nawiazania komunikacji
// zamiania na double 
      L     #iw_Nr_Rekordu;
      L     2;
      *I;
      ITD;
      SLD   3;
      T     #L_DW_Licznik_Rekordow;
//Transmisja
      A     #o_Przesylanie_Danych;
      JCN   et_4;
      L     DBW [#L_DW_Licznik_Rekordow];
      T     #ow_Kanal_Pobierania;
      L     #iw_Nr_Rekordu;
      T     #ow_Rekord_Powracajacy;
et_4: NOP   0;
end:  NOP   0;
NETWORK
TITLE =
//Zapis bitow przejsciowych
      L     LW 0;
      T     #io_Help_Word;
      BEU;
END_FUNCTION

DATA_BLOCK "Blok_Bledow"	// DB 119
VERSION : 0.1
  STRUCT
   Bledy : STRUCT
    Przek_Bezp_Nie_Ok : BOOL ;	//Blad przekanika bezpieczenstwa [I4.1 s. 10]
    Blad_Kom_Odbieranie : BOOL ;	//Blad komunikacji z odbieraniem [FC119]
    Bezpieczniki_Nie_Ok : BOOL ;	//Wyzwolenie wylacznika termicznego [I4.0 s. 10]
    Mayser_Nie_Ok : BOOL ;	//Wyzwolenie listwy bezpieczenstwa [I4.2 s.10]
    Foto_Zle_Pokrycie : BOOL ;	//Niedozwolone pokrycie fotokomorek obecnosci palety [I5.2,I5.3 s.11]
    Hamulec_Reczny_Rewizja : BOOL ;	//Hamulec reczny odbezpieczony [I5.6 s 11]
    Skaner_Wym_Przod_Reset : BOOL ;	//Skaner przod wymagany reset [I6.1 s.12]
    Skaner_Przod_Error : BOOL ;	//Blad Skanera przedniego lub jego  zabrudzenie [I6.2 s.12]
    Skaner_Przod_Strefa : BOOL ;	//Skaner przedni strefa wyzwolona I[I6.3 s.12]
    Skaner_Wym_Tyl_Reset : BOOL ;	//Skaner tylni wymagany reset [I7.1 s.12]
    Skaner_Tyl_Error : BOOL ;	//Blad Skanera tylniego lub jego  zabrudzenie [I7.2 s.12]
    Skaner_Tyl_Strefa : BOOL ;	//Skaner tylni strefa wyzwolona [I7.3 s.12]
    Obwody_Zew_Nie_Ok : BOOL ;	//Obwody bezpieczenstwa zewnetrzne nie Ok [I8.1 s.14](Not-Aus Slupy)
    Falownik_Sew_Blad : BOOL ;	//Blad falownika SEW [FC101]
    Falownik_Sew_N_Ready : BOOL ;	//Falownik sew nie gotowy [FC101]
    Falownik_Lenze_Blad : BOOL ;	//Blad falownika Lenze [FC101]
    Warunki_Startu_N_OK : BOOL ;	//Warunki startu Sew nie spelnione [FC101]
    Blad_Zwolnienia : BOOL ;	//Blad zwolnienia tasmy transportera [FC30]
    Help_int : INT ;	//Rezerwa dla booli
    Nr_Bledu_Sew : INT ;	//Blad specyficzny sew do odczytania
    Prad_Aktualny : INT ;	//Prad aktualny SEW [FC101]
    Predkosc_Aktualna : INT ;	//Predkosc akutualna wozka [FC101]
    Reserwa_Int : INT ;
    REserwa_Int1 : INT ;
   END_STRUCT ;
  END_STRUCT ;	
BEGIN
END_DATA_BLOCK

DATA_BLOCK "COM_ODB"	// DB 200
VERSION : 0.1
  STRUCT
   OUT : STRUCT
    Bit_Kom_Shuttle : BOOL ;	//Bit toggle komunikacji z wozkiem (<--)Shuttle
    Petla_Bezp_0_OK : BOOL ;	//Petla bezpieczenstwa 0 OK (<--Shuttle )
    Petla_Bezp_1_OK : BOOL ;	//Petla bezpieczenstwa 1 OK ( <--Shuttle)
    Wozek_Auto_Info : BOOL ;	//Wozek w Auto - 1 lub Reczny - 2
    Blad_Wozka : BOOL ;	//Wozek jest w bledzie
    Falownik_Band_Gotowy : BOOL ;	//Falownik Band Gotowy
    PB_Reset : BOOL ;	//Przycisk reset do grzybow na slupach
    Res_0_7 : BOOL ;
    Bit_Com_od_Shuttle : BOOL ;
    Potw_Nowej_Pozycji : BOOL ;	//Bit potwierdzenia przyjecia nowej pozycji (<-- Shuttle )
    Shuttle_Na_Pozycji : BOOL ;	//Wozek na pozycji (<--Shuttle )
    Shuttle_Stoi : BOOL ;	//Wozek na pozycji (Shuttle <--)
    Potw_Zasprz : BOOL ;	//Potwierdzenie zasprzeglenia (<--)Shuttle
    Potw_Rozprz : BOOL ;	//Potwierdzenie Rozprzeglenia (<--Shuttle )
    Foto_Przod : BOOL ;	//Fotokomorka wozek przod (<--Shuttle )
    Foto_Wozek_Tyl : BOOL ;	//Fotokomorka wozek tyl (<--Shuttle)
    Res_2_0 : BOOL ;
    Res_2_1 : BOOL ;
    Res_2_2 : BOOL ;
    Res_2_3 : BOOL ;
    Res_2_4 : BOOL ;
    Res_2_5 : BOOL ;
    Res_2_6 : BOOL ;
    Res_2_7 : BOOL ;
    Wybrana_Strefa_1_Przod : BOOL ;	//Strefa 1 Skaner Przod (<--Shuttle)
    Wybrana_Strefa_2_Przod : BOOL ;	//Strefa 2 Skaner Przod (<--Shuttle)
    Wybrana_Strefa_3_Przod : BOOL ;	//Strefa 3 Skaner Przod (<--Shuttle)
    Wybrana_Strefa_4_Przod : BOOL ;	//Strefa 4 Skaner Przod (<--Shuttle)
    Wybrana_Strefa_1_Tyl : BOOL ;	//Strefa 1 Skaner Tyl(<--Shuttle)
    Wybrana_Strefa_2_Tyl : BOOL ;	//Strefa 2 Skaner Tyl (<--Shuttle)
    Wybrana_Strefa_3_Tyl : BOOL ;	//Strefa 3 Skaner Tyl (<--Shuttle)
    Wybrana_Strefa_4_Tyl : BOOL ;	//Strefa 4 Skaner Tyl (<--Shuttle)
    Poz_Akt_Wozka : DINT ;	//Pozycja aktualna wozka
   END_STRUCT ;
   IN : STRUCT
    Bit_Kom_Odbieranie : BOOL ;	//Bit komunikacji do Shuttle(-->Shuttle)
    Bit_Bezpieczenstwa_0 : BOOL ;	//Bit bezpieczenstwa 0 (-->Shuttle)
    Reset_Wozka : BOOL ;	//Bit Resetu Shuttle ( -->Shuttle)
    Wozek_Auto : BOOL ;	//Bit ustawienia wozka Auto
    Wozek_Reczny : BOOL ;	//Bit ustwienia Reczny
    Partner_Reczny : BOOL ;	//Partner jest w recznym i wozek przyjmuje to
    Reset_Zadania : BOOL ;	//Reset zadania wozka
    Res_0_7 : BOOL ;
    Bit_Com_do_Shuttle : BOOL ;
    Bit_Nowej_Pozycji : BOOL ;	//Bit zadania nowej pozycji (-->Shuttle)
    Potw_Pozycji : BOOL ;	//Bit potwierdzenia pozycji (-->Shuttle)
    Rez_1_3 : BOOL ;
    Zasprz_Wozka : BOOL ;	//Rozkaz Zasprzeglenie Wozka (-->Shuttle)
    Rozprz_Wozka : BOOL ;	//Rozkaz Rozprzeglenie Wozka (--> Shuttle)
    Silnik_Banda_Lewo : BOOL ;	//Jazda silnika w lewo (-->Shuttle)
    Silnik_Banda_Prawo : BOOL ;	//Jazda silnika w prawo (-->Shuttle)
    Res_2_0 : BOOL ;
    Res_2_1 : BOOL ;
    Res_2_2 : BOOL ;
    Res_2_3 : BOOL ;
    Res_2_4 : BOOL ;
    Res_2_5 : BOOL ;
    Res_2_6 : BOOL ;
    Res_2_7 : BOOL ;
    Pozycja_KB1 : BOOL ;	//Blokada dalekiej jazdy w prawo
    Pozycja_KB2 : BOOL ;	//Blokada dalekiej jazdy w prawo
    Pozycja_Gender : BOOL ;	//Blokada dalekiej jazdy w lewo
    Pozycja_Intro_Pob : BOOL ;	//Blokada dalekiej jazdy w lewo
    Pozycja_Intro_Odb : BOOL ;	//Blokada dalekiej jazdy w lewo
    Res_3_5 : BOOL ;
    Res_3_6 : BOOL ;
    Res_3_7 : BOOL ;
    Pozycja_Zadana : DINT ;	//Pozycja zadana w mm (--> Shuttle)
   END_STRUCT ;
   SOME_OUT : STRUCT
    tab_32 : ARRAY  [1 .. 32 ] OF BYTE ;
   END_STRUCT ;
   SOME_IN : STRUCT
    tab_32 : ARRAY  [1 .. 32 ] OF BYTE ;
   END_STRUCT ;
  END_STRUCT ;	
BEGIN
END_DATA_BLOCK

DATA_BLOCK "LIN"	// DB 201
VERSION : 0.1
  STRUCT
   IN : STRUCT 	//Dane wejsciowe z Odbierania
    Zadanie_Transmisji : BOOL ;
    Zadanie_Danych : BOOL ;
    Toggle : BOOL ;	//bit- in/out
    Rezerwa_0_3 : BOOL ;
    Rezerwa_0_4 : BOOL ;
    Funcja_Receive : BOOL ;
    Funkcja_Share : BOOL ;
    Rezerwa_0_7 : BOOL ;
    Rezerwa_Bajt_1 : BYTE ;
    Nr_Bloku : INT  := 701;	//Nr bloku gdzie dane (read/send)
    Nr_Rekordu : INT ;	//Nr rekordu wysylanego (read/send)
    Kanal_Nadawania : INT ;	//Kanal Nadawania (send)
    Rezerwa_Bajtow : ARRAY  [1 .. 8 ] OF BYTE ;
    Predkosc_Cargo : INT  := 100;	//Predkosc Cargo w procentach
    Reserwa_Dalej : ARRAY  [1 .. 14 ] OF BYTE ;
   END_STRUCT ;
  END_STRUCT ;	
BEGIN
   IN.Nr_Bloku := 701;
   IN.Predkosc_Cargo := 100;
END_DATA_BLOCK

DATA_BLOCK "LOUT"	// DB 202
VERSION : 0.1
  STRUCT
   OUT : STRUCT 	//Dane wejsciowe z Odbierania
    Transmisja_Ustanowiona : BOOL ;
    Blok_Zarezerwowany : BOOL ;
    Toggle : BOOL ;	//bit- in/out
    Przesylanie_Danych : BOOL ;
    Koniec_Nadawania : BOOL ;
    Receive_Wybrane : BOOL ;
    Share_Wybrane : BOOL ;
    Rezerwa_0_7 : BOOL ;
    Rezerwa_Bajt_1 : BYTE ;
    Nr_Rekordu : INT  := 701;
    Licznik_Rekordow : INT ;	//Potwierdzenie Rekordu (Share/receive)
    Kanal_Pobierania : INT ;	//Pobieranie danych (Share)
    Rezerwa_Bajtow : ARRAY  [1 .. 8 ] OF BYTE ;
    Bledy : STRUCT
     Bledy_W_Bajtach : ARRAY  [1 .. 16 ] OF BYTE ;
    END_STRUCT ;
   END_STRUCT ;
  END_STRUCT ;	
BEGIN
   OUT.Nr_Rekordu := 701;
END_DATA_BLOCK

DATA_BLOCK "Blok_Parametrow"	// DB 701
VERSION : 0.1
  STRUCT
   Predkosc_Ostrzegawcza : DINT  := L#50;	//Zmiana predkosci procentowa w strefie ostrzegawczej [50]
   Predkosc_Maksymalna : DINT  := L#300;	//Predkosc maksymalna wozka
   Rampa_Startu_Wozka : DINT  := L#2000;	//Rampa startu wozka [ms]
   Rampa_Stopu_Wozka : DINT  := L#2000;	//Rampa stopu wozka [ms]
   Predkosc_Na_Pelno : DINT  := L#100;	//Predkosc w % wozka pelnego
   DB_VAR3 : DINT  := L#2;	//Temporary placeholder variable
   DB_VAR4 : DINT ;	//Temporary placeholder variable
   DB_VAR5 : DINT ;	//Temporary placeholder variable
   DB_VAR6 : DINT ;	//Temporary placeholder variable
   DB_VAR7 : DINT ;	//Temporary placeholder variable
   DB_VAR8 : DINT ;	//Temporary placeholder variable
   DB_VAR9 : DINT ;	//Temporary placeholder variable
   DB_VAR10 : DINT ;	//Temporary placeholder variable
   DB_VAR11 : DINT ;	//Temporary placeholder variable
   DB_VAR12 : DINT ;	//Temporary placeholder variable
   DB_VAR13 : DINT ;	//Temporary placeholder variable
   DB_VAR14 : DINT ;	//Temporary placeholder variable
   DB_VAR15 : DINT ;	//Temporary placeholder variable
   DB_VAR16 : DINT ;	//Temporary placeholder variable
   DB_VAR17 : DINT ;	//Temporary placeholder variable
   DB_VAR18 : DINT ;	//Temporary placeholder variable
   DB_VAR19 : DINT ;	//Temporary placeholder variable
   DB_VAR191 : DINT ;	//Temporary placeholder variable
   DB_VAR192 : DINT ;	//Temporary placeholder variable
   DB_VAR193 : DINT ;	//Temporary placeholder variable
   DB_VAR194 : DINT ;	//Temporary placeholder variable
   DB_VAR195 : DINT ;	//Temporary placeholder variable
   DB_VAR1951 : DINT ;	//Temporary placeholder variable
   DB_VAR19511 : DINT ;	//Temporary placeholder variable
   DB_VAR19512 : DINT ;	//Temporary placeholder variable
   DB_VAR19513 : DINT ;	//Temporary placeholder variable
   DB_VAR19514 : DINT ;	//Temporary placeholder variable
   DB_VAR19515 : DINT ;	//Temporary placeholder variable
   DB_VAR19516 : DINT ;	//Temporary placeholder variable
   DB_VAR19517 : DINT ;	//Temporary placeholder variable
   DB_VAR19518 : DINT ;	//Temporary placeholder variable
   DB_VAR19519 : DINT ;	//Temporary placeholder variable
   DB_VAR195110 : DINT ;	//Temporary placeholder variable
   DB_VAR195111 : DINT ;	//Temporary placeholder variable
   DB_VAR195112 : DINT ;	//Temporary placeholder variable
   DB_VAR195113 : DINT ;	//Temporary placeholder variable
   DB_VAR195114 : DINT ;	//Temporary placeholder variable
   DB_VAR195115 : DINT ;	//Temporary placeholder variable
   DB_VAR195116 : DINT ;	//Temporary placeholder variable
   DB_VAR195117 : DINT ;	//Temporary placeholder variable
   DB_VAR195118 : DINT ;	//Temporary placeholder variable
   DB_VAR195119 : DINT ;	//Temporary placeholder variable
   DB_VAR195120 : DINT ;	//Temporary placeholder variable
   DB_VAR195121 : DINT ;	//Temporary placeholder variable
   DB_VAR195122 : DINT ;	//Temporary placeholder variable
  END_STRUCT ;	
BEGIN
   Predkosc_Ostrzegawcza := L#30;
   Predkosc_Maksymalna := L#500;
   Rampa_Startu_Wozka := L#2000;
   Rampa_Stopu_Wozka := L#2000;
   Predkosc_Na_Pelno := L#80;
   DB_VAR3 := L#2;
END_DATA_BLOCK

DATA_BLOCK "Blok_Stref_Kier_KB1"	// DB 720
VERSION : 0.1
  STRUCT
   Wartosc_Poz_Kier_KB1 : STRUCT 	//Wartosc pozycji
    Poz_0 : DINT  := L#37000;
    Poz_1 : DINT  := L#33000;
    Poz_2 : DINT  := L#17000;
    Poz_3 : DINT  := L#12000;
    Poz_4 : DINT  := L#9000;
    Poz_5 : DINT  := L#5000;
    Poz_6 : DINT  := L#20;
    Poz_7 : DINT ;
    Poz_8 : DINT ;
    Poz_9 : DINT ;
    Poz_10 : DINT ;
    Poz_11 : DINT ;
    Poz_12 : DINT ;
    poz_13 : DINT ;
    Poz_14 : DINT ;
    Poz_15 : DINT ;
    Poz_16 : DINT ;
    Poz_17 : DINT ;
    Poz_18 : DINT ;
    Poz_19 : DINT ;
    Poz_20 : DINT ;
    Poz_21 : DINT ;
    Poz_22 : DINT ;
    poz_23 : DINT ;
    Poz_24 : DINT ;
   END_STRUCT ;
   Wartosc_Strefy : STRUCT 	//Wartosc Strefy
    Strefa_0 : DINT  := L#4;
    Strefa_1 : DINT  := L#4;
    Strefa_2 : DINT  := L#4;
    Strefa_3 : DINT  := L#4;
    Strefa_4 : DINT  := L#4;
    Strefa_5 : DINT  := L#4;
    Strefa_6 : DINT  := L#4;
    Strefa_7 : DINT  := L#4;
    Strefa_8 : DINT  := L#4;
    Strefa_9 : DINT  := L#4;
    Strefa_10 : DINT  := L#4;
    Strefa_11 : DINT  := L#4;
    Strefa_12 : DINT  := L#4;
    Strefa_13 : DINT  := L#4;
    Strefa_14 : DINT  := L#4;
    Strefa_15 : DINT  := L#4;
    Strefa_16 : DINT  := L#4;
    Strefa_17 : DINT  := L#4;
    Strefa_18 : DINT  := L#4;
    Strefa_19 : DINT  := L#4;
    Strefa_20 : DINT  := L#4;
    Strefa_21 : DINT  := L#4;
    Strefa_22 : DINT  := L#4;
    Strefa_23 : DINT  := L#4;
    Strefa_24 : DINT  := L#4;
   END_STRUCT ;
   Wartosc_Predkosci : STRUCT 	//Wartosc Predkosci w procentach
    Predkosc_0 : DINT  := L#100;
    Predkosc_1 : DINT  := L#100;
    Predkosc_2 : DINT  := L#100;
    Predkosc_3 : DINT  := L#100;
    Predkosc_4 : DINT  := L#100;
    Predkosc_5 : DINT  := L#100;
    Predkosc_6 : DINT  := L#100;
    Predkosc_7 : DINT  := L#100;
    Predkosc_8 : DINT  := L#100;
    Predkosc_9 : DINT  := L#100;
    Predkosc_10 : DINT  := L#100;
    Predkosc_11 : DINT  := L#100;
    Predkosc_12 : DINT  := L#100;
    Predkosc_13 : DINT  := L#100;
    Predkosc_14 : DINT  := L#100;
    Predkosc_15 : DINT  := L#100;
    Predkosc_16 : DINT  := L#100;
    Predkosc_17 : DINT  := L#100;
    Predkosc_18 : DINT  := L#100;
    Predkosc_19 : DINT  := L#100;
    Predkosc_20 : DINT  := L#100;
    Predkosc_21 : DINT  := L#100;
    Predkosc_22 : DINT  := L#100;
    Predkosc_23 : DINT  := L#100;
    Predkosc_24 : DINT  := L#100;
   END_STRUCT ;
  END_STRUCT ;	
BEGIN
   Wartosc_Poz_Kier_KB1.Poz_0 := L#37000;
   Wartosc_Poz_Kier_KB1.Poz_1 := L#33000;
   Wartosc_Poz_Kier_KB1.Poz_2 := L#17000;
   Wartosc_Poz_Kier_KB1.Poz_3 := L#12000;
   Wartosc_Poz_Kier_KB1.Poz_4 := L#9000;
   Wartosc_Poz_Kier_KB1.Poz_5 := L#5000;
   Wartosc_Poz_Kier_KB1.Poz_6 := L#20;
   Wartosc_Strefy.Strefa_0 := L#1;
   Wartosc_Strefy.Strefa_1 := L#2;
   Wartosc_Strefy.Strefa_2 := L#4;
   Wartosc_Strefy.Strefa_3 := L#3;
   Wartosc_Strefy.Strefa_4 := L#2;
   Wartosc_Strefy.Strefa_5 := L#1;
   Wartosc_Strefy.Strefa_6 := L#3;
   Wartosc_Strefy.Strefa_7 := L#4;
   Wartosc_Strefy.Strefa_8 := L#4;
   Wartosc_Strefy.Strefa_9 := L#4;
   Wartosc_Strefy.Strefa_10 := L#4;
   Wartosc_Strefy.Strefa_11 := L#4;
   Wartosc_Strefy.Strefa_12 := L#4;
   Wartosc_Strefy.Strefa_13 := L#4;
   Wartosc_Strefy.Strefa_14 := L#4;
   Wartosc_Strefy.Strefa_15 := L#4;
   Wartosc_Strefy.Strefa_16 := L#4;
   Wartosc_Strefy.Strefa_17 := L#4;
   Wartosc_Strefy.Strefa_18 := L#4;
   Wartosc_Strefy.Strefa_19 := L#4;
   Wartosc_Strefy.Strefa_20 := L#4;
   Wartosc_Strefy.Strefa_21 := L#4;
   Wartosc_Strefy.Strefa_22 := L#4;
   Wartosc_Strefy.Strefa_23 := L#4;
   Wartosc_Strefy.Strefa_24 := L#4;
   Wartosc_Predkosci.Predkosc_0 := L#100;
   Wartosc_Predkosci.Predkosc_1 := L#100;
   Wartosc_Predkosci.Predkosc_2 := L#100;
   Wartosc_Predkosci.Predkosc_3 := L#100;
   Wartosc_Predkosci.Predkosc_4 := L#100;
   Wartosc_Predkosci.Predkosc_5 := L#100;
   Wartosc_Predkosci.Predkosc_6 := L#100;
   Wartosc_Predkosci.Predkosc_7 := L#100;
   Wartosc_Predkosci.Predkosc_8 := L#100;
   Wartosc_Predkosci.Predkosc_9 := L#100;
   Wartosc_Predkosci.Predkosc_10 := L#100;
   Wartosc_Predkosci.Predkosc_11 := L#100;
   Wartosc_Predkosci.Predkosc_12 := L#100;
   Wartosc_Predkosci.Predkosc_13 := L#100;
   Wartosc_Predkosci.Predkosc_14 := L#100;
   Wartosc_Predkosci.Predkosc_15 := L#100;
   Wartosc_Predkosci.Predkosc_16 := L#100;
   Wartosc_Predkosci.Predkosc_17 := L#100;
   Wartosc_Predkosci.Predkosc_18 := L#100;
   Wartosc_Predkosci.Predkosc_19 := L#100;
   Wartosc_Predkosci.Predkosc_20 := L#100;
   Wartosc_Predkosci.Predkosc_21 := L#100;
   Wartosc_Predkosci.Predkosc_22 := L#100;
   Wartosc_Predkosci.Predkosc_23 := L#100;
   Wartosc_Predkosci.Predkosc_24 := L#100;
END_DATA_BLOCK

DATA_BLOCK "Blok_Stref_Kier_Rot"	// DB 721
VERSION : 0.1
  STRUCT
   Wartosc_Pozycji : STRUCT 	//Wartosc pozycji
    Poz_0 : DINT ;
    Poz_1 : DINT  := L#1000;
    Poz_2 : DINT  := L#2000;
    Poz_3 : DINT  := L#5000;
    Poz_4 : DINT  := L#20000;
    Poz_5 : DINT  := L#40000;
    Poz_6 : DINT ;
    Poz_7 : DINT ;
    Poz_8 : DINT ;
    Poz_9 : DINT ;
    Poz_10 : DINT ;
    Poz_11 : DINT ;
    Poz_12 : DINT ;
    poz_13 : DINT ;
    Poz_14 : DINT ;
    Poz_15 : DINT ;
    Poz_16 : DINT ;
    Poz_17 : DINT ;
    Poz_18 : DINT ;
    Poz_19 : DINT ;
    Poz_20 : DINT ;
    Poz_21 : DINT ;
    Poz_22 : DINT ;
    poz_23 : DINT ;
    Poz_24 : DINT ;
   END_STRUCT ;
   Wartosc_Strefy : STRUCT 	//Wartosc Strefy
    Strefa_0 : DINT  := L#4;
    Strefa_1 : DINT  := L#4;
    Strefa_2 : DINT  := L#4;
    Strefa_3 : DINT  := L#3;
    Strefa_4 : DINT  := L#4;
    Strefa_5 : DINT  := L#4;
    Strefa_6 : DINT  := L#4;
    Strefa_7 : DINT  := L#4;
    Strefa_8 : DINT  := L#4;
    Strefa_9 : DINT  := L#4;
    Strefa_10 : DINT  := L#4;
    Strefa_11 : DINT  := L#4;
    Strefa_12 : DINT  := L#4;
    Strefa_13 : DINT  := L#4;
    Strefa_14 : DINT  := L#4;
    Strefa_15 : DINT  := L#4;
    Strefa_16 : DINT  := L#4;
    Strefa_17 : DINT  := L#4;
    Strefa_18 : DINT  := L#4;
    Strefa_19 : DINT  := L#4;
    Strefa_20 : DINT  := L#4;
    Strefa_21 : DINT  := L#4;
    Strefa_22 : DINT  := L#4;
    Strefa_23 : DINT  := L#4;
    Strefa_24 : DINT  := L#4;
   END_STRUCT ;
   Wartosc_Predkosci : STRUCT 	//Wartosc Predkosci w procentach
    Predkosc_0 : DINT  := L#100;
    Predkosc_1 : DINT  := L#100;
    Predkosc_2 : DINT  := L#100;
    Predkosc_3 : DINT  := L#100;
    Predkosc_4 : DINT  := L#100;
    Predkosc_5 : DINT  := L#100;
    Predkosc_6 : DINT  := L#100;
    Predkosc_7 : DINT  := L#100;
    Predkosc_8 : DINT  := L#100;
    Predkosc_9 : DINT  := L#100;
    Predkosc_10 : DINT  := L#100;
    Predkosc_11 : DINT  := L#100;
    Predkosc_12 : DINT  := L#100;
    Predkosc_13 : DINT  := L#100;
    Predkosc_14 : DINT  := L#100;
    Predkosc_15 : DINT  := L#100;
    Predkosc_16 : DINT  := L#100;
    Predkosc_17 : DINT  := L#100;
    Predkosc_18 : DINT  := L#100;
    Predkosc_19 : DINT  := L#100;
    Predkosc_20 : DINT  := L#100;
    Predkosc_21 : DINT  := L#100;
    Predkosc_22 : DINT  := L#100;
    Predkosc_23 : DINT  := L#100;
    Predkosc_24 : DINT  := L#100;
   END_STRUCT ;
  END_STRUCT ;	
BEGIN
   Wartosc_Pozycji.Poz_0 := L#40;
   Wartosc_Pozycji.Poz_1 := L#1000;
   Wartosc_Pozycji.Poz_2 := L#2000;
   Wartosc_Pozycji.Poz_3 := L#7020;
   Wartosc_Pozycji.Poz_4 := L#29000;
   Wartosc_Pozycji.Poz_5 := L#30000;
   Wartosc_Pozycji.Poz_6 := L#40000;
   Wartosc_Strefy.Strefa_0 := L#1;
   Wartosc_Strefy.Strefa_1 := L#2;
   Wartosc_Strefy.Strefa_2 := L#3;
   Wartosc_Strefy.Strefa_3 := L#2;
   Wartosc_Strefy.Strefa_4 := L#1;
   Wartosc_Strefy.Strefa_5 := L#4;
   Wartosc_Strefy.Strefa_6 := L#4;
   Wartosc_Strefy.Strefa_7 := L#4;
   Wartosc_Strefy.Strefa_8 := L#4;
   Wartosc_Strefy.Strefa_9 := L#4;
   Wartosc_Strefy.Strefa_10 := L#4;
   Wartosc_Strefy.Strefa_11 := L#4;
   Wartosc_Strefy.Strefa_12 := L#4;
   Wartosc_Strefy.Strefa_13 := L#4;
   Wartosc_Strefy.Strefa_14 := L#4;
   Wartosc_Strefy.Strefa_15 := L#4;
   Wartosc_Strefy.Strefa_16 := L#4;
   Wartosc_Strefy.Strefa_17 := L#4;
   Wartosc_Strefy.Strefa_18 := L#4;
   Wartosc_Strefy.Strefa_19 := L#4;
   Wartosc_Strefy.Strefa_20 := L#4;
   Wartosc_Strefy.Strefa_21 := L#4;
   Wartosc_Strefy.Strefa_22 := L#4;
   Wartosc_Strefy.Strefa_23 := L#4;
   Wartosc_Strefy.Strefa_24 := L#4;
   Wartosc_Predkosci.Predkosc_0 := L#100;
   Wartosc_Predkosci.Predkosc_1 := L#100;
   Wartosc_Predkosci.Predkosc_2 := L#100;
   Wartosc_Predkosci.Predkosc_3 := L#100;
   Wartosc_Predkosci.Predkosc_4 := L#100;
   Wartosc_Predkosci.Predkosc_5 := L#100;
   Wartosc_Predkosci.Predkosc_6 := L#100;
   Wartosc_Predkosci.Predkosc_7 := L#100;
   Wartosc_Predkosci.Predkosc_8 := L#100;
   Wartosc_Predkosci.Predkosc_9 := L#100;
   Wartosc_Predkosci.Predkosc_10 := L#100;
   Wartosc_Predkosci.Predkosc_11 := L#100;
   Wartosc_Predkosci.Predkosc_12 := L#100;
   Wartosc_Predkosci.Predkosc_13 := L#100;
   Wartosc_Predkosci.Predkosc_14 := L#100;
   Wartosc_Predkosci.Predkosc_15 := L#100;
   Wartosc_Predkosci.Predkosc_16 := L#100;
   Wartosc_Predkosci.Predkosc_17 := L#100;
   Wartosc_Predkosci.Predkosc_18 := L#100;
   Wartosc_Predkosci.Predkosc_19 := L#100;
   Wartosc_Predkosci.Predkosc_20 := L#100;
   Wartosc_Predkosci.Predkosc_21 := L#100;
   Wartosc_Predkosci.Predkosc_22 := L#100;
   Wartosc_Predkosci.Predkosc_23 := L#100;
   Wartosc_Predkosci.Predkosc_24 := L#100;
END_DATA_BLOCK

ORGANIZATION_BLOCK "Program_Glowny"	// OB 1
VERSION : 0.1
VAR_TEMP
  OB1_EV_CLASS : BYTE ;	//Bits 0-3 = 1 (Coming event), Bits 4-7 = 1 (Event class 1)
  OB1_SCAN_1 : BYTE ;	//1 (Cold restart scan 1 of OB 1), 3 (Scan 2-n of OB 1)
  OB1_PRIORITY : BYTE ;	//1 (Priority of 1 is lowest)
  OB1_OB_NUMBR : BYTE ;	//1 (Organization block 1, OB1)
  OB1_RESERVED_1 : BYTE ;	//Reserved for system
  OB1_RESERVED_2 : BYTE ;	//Reserved for system
  OB1_PREV_CYCLE : INT ;	//Cycle time of previous OB1 scan (milliseconds)
  OB1_MIN_CYCLE : INT ;	//Minimum cycle time of OB1 (milliseconds)
  OB1_MAX_CYCLE : INT ;	//Maximum cycle time of OB1 (milliseconds)
  OB1_DATE_TIME : DATE_AND_TIME ;	//Date and time OB1 started
  SERVICE : INT ;
END_VAR
BEGIN
NETWORK
TITLE = Sprungverteiler
//Ten Network celowo jest wolny
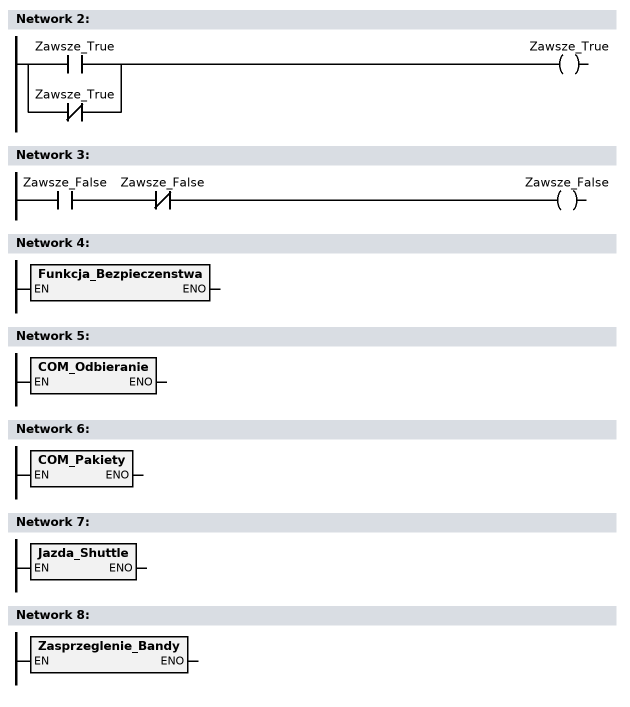
NETWORK
TITLE =
//Marka globalna zawsze 1 
      O     "Zawsze_True";
      ON    "Zawsze_True";
      =     "Zawsze_True";
NETWORK
TITLE =
//Marka globalna zawsze 0
      A     "Zawsze_False";
      AN    "Zawsze_False";
      =     "Zawsze_False";
NETWORK
TITLE =
//wyolanie funkcji bezpieczenstwa
      CALL  "Funkcja_Bezpieczenstwa";
      NOP   0;
NETWORK
TITLE =
      CALL  "COM_Odbieranie";
      NOP   0;
NETWORK
TITLE =
      CALL  "COM_Pakiety";
      NOP   0;
NETWORK
TITLE =
//Wywolanie funcji obslugi wozka
//
      CALL  "Jazda_Shuttle";
      NOP   0;
NETWORK
TITLE =
//Obsluga bandy jezdzacej
      CALL  "Zasprzeglenie_Bandy";
      NOP   0;
END_ORGANIZATION_BLOCK

ORGANIZATION_BLOCK "I/O_FLT1"	// OB 82
TITLE = "I/O Point Fault"
VERSION : 0.1
VAR_TEMP
  OB82_EV_CLASS : BYTE ;	//16#39, Event class 3, Entering event state, Internal fault event
  OB82_FLT_ID : BYTE ;	//16#XX, Fault identifcation code
  OB82_PRIORITY : BYTE ;	//Priority of OB Execution
  OB82_OB_NUMBR : BYTE ;	//82 (Organization block 82, OB82)
  OB82_RESERVED_1 : BYTE ;	//Reserved for system
  OB82_IO_FLAG : BYTE ;	//Input (01010100), Output (01010101)
  OB82_MDL_ADDR : WORD ;	//Base address of module with fault
  OB82_MDL_DEFECT : BOOL ;	//Module defective
  OB82_INT_FAULT : BOOL ;	//Internal fault
  OB82_EXT_FAULT : BOOL ;	//External fault
  OB82_PNT_INFO : BOOL ;	//Point information
  OB82_EXT_VOLTAGE : BOOL ;	//External voltage low
  OB82_FLD_CONNCTR : BOOL ;	//Field wiring connector missing
  OB82_NO_CONFIG : BOOL ;	//Module has no configuration data
  OB82_CONFIG_ERR : BOOL ;	//Module has configuration error
  OB82_MDL_TYPE : BYTE ;	//Type of module
  OB82_SUB_MDL_ERR : BOOL ;	//Sub-Module is missing or has error
  OB82_COMM_FAULT : BOOL ;	//Communication fault
  OB82_MDL_STOP : BOOL ;	//Module is stopped
  OB82_WTCH_DOG_FLT : BOOL ;	//Watch dog timer stopped module
  OB82_INT_PS_FLT : BOOL ;	//Internal power supply fault
  OB82_PRIM_BATT_FLT : BOOL ;	//Primary battery is in fault
  OB82_BCKUP_BATT_FLT : BOOL ;	//Backup battery is in fault
  OB82_RESERVED_2 : BOOL ;	//Reserved for system
  OB82_RACK_FLT : BOOL ;	//Rack fault, only for bus interface module
  OB82_PROC_FLT : BOOL ;	//Processor fault
  OB82_EPROM_FLT : BOOL ;	//EPROM fault
  OB82_RAM_FLT : BOOL ;	//RAM fault
  OB82_ADU_FLT : BOOL ;	//ADU fault
  OB82_FUSE_FLT : BOOL ;	//Fuse fault
  OB82_HW_INTR_FLT : BOOL ;	//Hardware interupt input in fault
  OB82_RESERVED_3 : BOOL ;	//Reserved for system
  OB82_DATE_TIME : DATE_AND_TIME ;	//Date and time OB82 started
END_VAR
BEGIN
// (block stored without names or comments; labels and parameter names are numbered)
END_ORGANIZATION_BLOCK

ORGANIZATION_BLOCK "RACK_FLT"	// OB 86
TITLE = "Loss Of Rack Fault"
VERSION : 0.1
VAR_TEMP
  OB86_EV_CLASS : BYTE ;	//16#38/39 Event class 3
  OB86_FLT_ID : BYTE ;	//16#C1/C4/C5, Fault identifcation code
  OB86_PRIORITY : BYTE ;	//Priority of OB Execution
  OB86_OB_NUMBR : BYTE ;	//86 (Organization block 86, OB86)
  OB86_RESERVED_1 : BYTE ;	//Reserved for system
  OB86_RESERVED_2 : BYTE ;	//Reserved for system
  OB86_MDL_ADDR : WORD ;	//Base address of IM module in rack with fault
  OB86_RACKS_FLTD : ARRAY  [0 .. 31 ] OF BOOL ;	//Racks in fault
  OB86_DATE_TIME : DATE_AND_TIME ;	//Date and time OB86 started
END_VAR
BEGIN
// (block stored without names or comments; labels and parameter names are numbered)
END_ORGANIZATION_BLOCK

ORGANIZATION_BLOCK "PROG_ERR"	// OB 121
TITLE = "Programming Error"
VERSION : 0.1
VAR_TEMP
  OB121_EV_CLASS : BYTE ;	//16#25, Event class 2, Entering event state, Internal fault event
  OB121_SW_FLT : BYTE ;	//16#XX Software programming fault
  OB121_PRIORITY : BYTE ;	//Priority of OB Execution
  OB121_OB_NUMBR : BYTE ;	//121 (Organization block 121, OB121)
  OB121_BLK_TYPE : BYTE ;	//16#88/8A/8B/8C/8E Type of block fault occured in
  OB121_RESERVED_1 : BYTE ;	//Reserved for system
  OB121_FLT_REG : WORD ;	//16#XX Specific register that caused fault
  OB121_BLK_NUM : WORD ;	//Number of block that programming fault occured in
  OB121_PRG_ADDR : WORD ;	//Address in block where programming fault occured
  OB121_DATE_TIME : DATE_AND_TIME ;	//Date and time OB121 started
END_VAR
BEGIN
// (block stored without names or comments; labels and parameter names are numbered)
END_ORGANIZATION_BLOCK

ORGANIZATION_BLOCK "MOD_ERR"	// OB 122
TITLE = "Module Access Error"
VERSION : 0.1
VAR_TEMP
  OB122_EV_CLASS : BYTE ;	//16#29, Event class 2, Entering event state, Internal fault event
  OB122_SW_FLT : BYTE ;	//16#XX Software error code
  OB122_PRIORITY : BYTE ;	//Priority of OB Execution
  OB122_OB_NUMBR : BYTE ;	//122 (Organization block 122, OB122)
  OB122_BLK_TYPE : BYTE ;	//16#88/8C/8E Type of block fault occured in
  OB122_MEM_AREA : BYTE ;	//Memory area where access error occured
  OB122_MEM_ADDR : WORD ;	//Memory address where access error occured
  OB122_BLK_NUM : WORD ;	//Block number in which error occured
  OB122_PRG_ADDR : WORD ;	//Program address where error occured
  OB122_DATE_TIME : DATE_AND_TIME ;	//Date and time OB1 started
END_VAR
BEGIN
// (block stored without names or comments; labels and parameter names are numbered)
END_ORGANIZATION_BLOCK

SYMBOL_TABLE
""		
"AIO"	DB 10	DB 10
"Blok_Para"	DB 12	DB 12
"Blok_Bledow_Program"	DB 13	DB 13
"Asi_input"	DB 80	DB 80
"Asi_output"	DB 81	DB 81
"MPI_GD"	DB 100	DB 100	// Blok wymiany danych po mpi
"Blok_Bledow"	DB 119	DB 119
"DB_HMI"	DB 120	DB 120	// Blok wejsc wyjsc HMI
"Data_I_Czas"	DB 205	DB 205
"TEST_OBR2"	FB 2	FB 2	// Test obrotnicy nr 2
"Czesc_Bindujaca"	FB 3	FB 3	// Blok jazdy band bindownicy
"Blok_Jazdy_Band"	FB 5	FB 5
"Filtr_zbocza_2"	FB 14	FB 14
"T_ON"	FB 20	FB 20	// Timer on delay with memory
"T_ON_+_RESET"	FB 21	FB 21	// Czasowka on delay z zapamietanym czasem  + reset
"Banda_Podwojna"	FB 29	FB 29
"Banda_Pojedyncza"	FB 30	FB 30
"Banda_Obr_1"	FB 31	FB 31	// Banda obrotowa o dwoch wlotach i jednej fotokomorce
"Banda_Obr_2"	FB 32	FB 32	// Banda obrotowa nr 2
"Banda_Poj_+Tryb_Reczny"	FB 33	FB 33
"Banda_Obr_Bind"	FB 34	FB 34	// Banda obrotowa sluzaca do bindowania
"Blok_Pracy_Bindownicy"	FB 35	FB 35	// funkcja pozycjonujaca bande
"Wybranie_Wjazdu"	FB 50	FB 50
"Obr_Na_Poz_1"	FB 51	FB 51
"Obr_Na_Poz_2"	FB 52	FB 52	// Obrot na pozycje uwzgledniajacy czujniki 45st
"Obr_Na_Poz_3"	FB 53	FB 53	// Funkcja sterujaca obrotem talerza 4 po³o¿enia.
"Obr_Na_Poz_4"	FB 54	FB 54
"Pozycjonowanie_Bandy"	FB 55	FB 55
"Poz_Band_Back"	FB 56	FB 56
"Bindownica_Test"	FB 57	FB 57	// Testowy blok wejsc wyjsc bindownicy
"Pozycjonowanie_Palety"	FB 58	FB 58	// Funkcja pozycjonujaca palete
"TSEND"	FB 63	FB 63	// Send Data
"TRCV"	FB 64	FB 64	// Receive Data
"Blok_kodow_Pracy"	FB 80	FB 80
"Funkcja_Bezpieczenstwa"	FC 3	FC 3
"Sprawdzenie_Czujnikow"	FC 4	FC 4
"Szukaj_Zmiany"	FC 5	FC 5	// Funkcja szukajaca zmiany w obszarze odwzorowania
"FC_Lampki"	FC 6	FC 6	// Funkcja sterujaca lampkami
"Szukaj_Zmiany_2"	FC 7	FC 7
"Toggle"	FC 8	FC 8	// Funkcja przycisku bistabilnego
"Sterwanie_Swiatlo"	FC 9	FC 9	// Sterowanie sygnalami swietlnymi
"Lampka_Blad"	FC 10	FC 10
"Przyporzadkowanie_Wejsc"	FC 20	FC 20
"Przyporzadkowanie_Wyjsc"	FC 21	FC 21
"Rejestr_Tasm"	FC 30	FC 30
"FC_Auto_Reczny"	FC 40	FC 40
"Przycisk_Reset"	FC 41	FC 41	// Kasowanie_Bledow
"Wybor_Wjazdu"	FC 50	FC 50	// Wybor miejsca pobierania palety
"Obrotnica_Na_Pozycje"	FC 51	FC 51
"ASI_Odczyt"	FC 80	FC 80
"ASI_Zapis"	FC 81	FC 81
"Opoznienie_Wylotu"	FC 85	FC 85
"Opoznienie_Wlotu"	FC 86	FC 86	// Funkcja opozniajaca wlot
"Opoznienie_Wlotu_2"	FC 87	FC 87
"Komunikacja_GD"	FC 100	FC 100	// Komunikacja szafa foliarka
"Obsluga bledow"	FC 119	FC 119	// funkcja przekazujaca bledy do bloku db
"FC_HMI"	FC 120	FC 120
"Step_Control"	FC 127	FC 127	// Kontrola krokow
"Inkrementacja_Kroku"	FC 128	FC 128	// Funkcja inkrementujaca kroku
"Step_Control_2"	FC 130	FC 130
"Utworz_Blad"	FC 132	FC 132	// Funkcja stwarz kod bledu
"Funkcja_Zegara"	FC 140	FC 140	// Funkcja zegara
"pb_Strefa_bezpieczenstwa"	I 0.0	BOOL
"pb_Reczny"	I 0.1	BOOL
"pb_Auto"	I 0.2	BOOL
"pb_Reset"	I 0.3	BOOL
"pb_Stop"	I 0.4	BOOL
"pb_Cykl_Start"	I 0.5	BOOL
"pb_Tasma_1_Tyl"	I 0.6	BOOL
"pb_Tasma_1_Przod"	I 0.7	BOOL
"pb_Tasma_2_Tyl"	I 1.0	BOOL
"pb_Tasma_2_Przod"	I 1.1	BOOL
"pb_Tasma_3_Tyl"	I 1.2	BOOL
"pb_Tasma_3_Przod"	I 1.3	BOOL
"pb_Tasma_4_Tyl"	I 1.4	BOOL
"pb_Tasma_4_Przod"	I 1.5	BOOL
"pb_Tasma_3_Obr_CW"	I 1.6	BOOL
"pb_Tasma_3_Obr_CCW"	I 1.7	BOOL
"Obwod_Bezp_Bindownicy"	I 2.0	BOOL
"Bind_Polozenie_Podst"	I 2.1	BOOL
"Blad_Bindownicy"	I 2.2	BOOL
"Start_Koniec_Wiazania"	I 2.3	BOOL
"Bindownica_Auto"	I 2.4	BOOL	// Bindownica jest w trybie automatyki
"rez_i_2_5"	I 2.5	BOOL
"Prasa_W_Gorze"	I 2.6	BOOL
"Foto_Wozek"	I 2.7	BOOL
"i_foto_lewo_1"	I 3.0	BOOL
"i_foto_lewo_2"	I 3.1	BOOL
"i_foto_prawo_1"	I 3.2	BOOL
"i_foto_prawo_2"	I 3.3	BOOL
"rez_i_3_4"	I 3.4	BOOL
"rez_i_3_5"	I 3.5	BOOL
"rez_i_3_6"	I 3.6	BOOL
"rez_i_3_7"	I 3.7	BOOL
"Przekaznik_Bezp_OK"	I 4.0	BOOL
"Start"	I 4.1	BOOL
"Stop"	I 4.2	BOOL
"Praca_Z_Etykietami"	I 4.3	BOOL
"Przek_Rejonu_Bind_Ok"	I 4.4	BOOL
"Silownik_Etyk_Tyl"	I 5.0	BOOL
"Etyk_Gotowa"	I 5.1	BOOL
"Dane_W_Drukarce"	I 5.2	BOOL
"Brak_Papieru"	I 5.3	BOOL
"Drukuj_Recznie"	I 5.4	BOOL
"Bity_Przyciskow"	IB 0	BYTE
"Zawsze_True"	M 0.0	BOOL
"Zawsze_False"	M 0.1	BOOL
"Help_Start"	M 1.0	BOOL
"Help_Zbocze_Start"	M 1.1	BOOL
"Help_Start_2"	M 1.2	BOOL
"Marka_Bezpieczenstwa"	M 2.0	BOOL
"Marka_Start_Stop"	M 2.1	BOOL
"Marka_Bezpieczenstwa_2"	M 2.2	BOOL
"Rejon_Bindownicy_Stop"	M 2.3	BOOL
"Strefa_Bind_Ok"	M 2.4	BOOL
"Help_PB_Stop"	M 2.5	BOOL
"Edge_2_6"	M 2.6	BOOL
"Freeze"	M 2.7	BOOL
"Brak_Bledu"	M 3.0	BOOL
"Falowniki_OK"	M 3.1	BOOL
"Fuse_OK"	M 3.2	BOOL
"Help_Freeze"	M 3.3	BOOL
"Marka_Bezpieczenstwa_3"	M 3.4	BOOL
"Zezwolenie_Na_Wjazd"	M 3.5	BOOL	// Do stawiania lini
"Stop_Hmi"	M 3.7	BOOL
"Not_Aus_27_OK"	M 4.0	BOOL
"Not_Aus_28_OK"	M 4.1	BOOL
"Not_Aus_29_OK"	M 4.2	BOOL
"Strefa_Bind_Zamk"	M 4.3	BOOL
"Not_Aus_30_OK"	M 4.4	BOOL
"Not_Aus_31_OK"	M 4.5	BOOL
"Zmiana_Wykryta"	M 5.0	BOOL
"Help_M5.1"	M 5.1	BOOL
"Cykl_Binowania_Przwyr"	M 5.2	BOOL
"Help_M5.3"	M 5.3	BOOL
"Help_M5.4"	M 5.4	BOOL
"Kat_Jazdy_Rolek_OK"	M 5.5	BOOL
"Kat_Obrotnicy_Bezp"	M 5.6	BOOL
"Kurtyny_Wlot_Ok"	M 6.0	BOOL
"Kurtyny_Wylot_Ok"	M 6.1	BOOL
"Rygiel_OK"	M 6.2	BOOL
"Wirtualny_Sygnal_Bezp"	M 6.3	BOOL
"M_Zez_Na_Prace_Bind"	M 6.4	BOOL
"M_Obwod_Bezp_Bind"	M 6.5	BOOL
"Help_M6.6"	M 6.6	BOOL
"Warunki_Startu_OK"	M 7.0	BOOL
"Help_Bit_M_7_1"	M 7.1	BOOL
"Pomoc_Reczny"	M 7.7	BOOL
"M_Blad_Cyklu_Bindowania"	M 8.0	BOOL	// Blad cyklu
"M_Trick"	M 8.1	BOOL
"M_Cykl_Bindowania_Trwa"	M 9.0	BOOL
"M_Reset_Bledow"	M 20.0	BOOL
"M_Reset_Krokow"	M 20.1	BOOL
"Help_M20.2"	M 20.2	BOOL
"M_Help_Reset_Bledow"	M 20.3	BOOL
"M_pb_Cykl_Start"	M 20.5	BOOL
"Auto_Sprawdzone"	M 20.6	BOOL
"M_Powrot_do_Stopu"	M 20.7	BOOL
"Brak_Bledow_Do_Auto"	M 21.0	BOOL	// Brak bledow przy pojsicu w auto
"Blad_Automatu"	M 21.1	BOOL	// Blad automatu
"Help_M21.2"	M 21.2	BOOL
"help_m21.3"	M 21.3	BOOL
"Edge_M22.0"	M 22.0	BOOL
"M_Foto_1_Banda_11"	M 30.0	BOOL
"M_Foto_1_Banda_14"	M 40.0	BOOL
"Help_M_40_1"	M 40.1	BOOL
"M_Foto_1_Tasma_1"	M 40.2	BOOL
"Help_M_40_3"	M 40.3	BOOL
"M_Foto_1_Banda_3"	M 40.4	BOOL
"Help_M_40_5"	M 40.5	BOOL
"M_Foto_1_Banda_12"	M 40.6	BOOL
"Help_M_40_7"	M 40.7	BOOL
"Help_Foto"	M 41.0	BOOL
"M_Foto_1_Banda_2"	M 41.1	BOOL
"Bini_Prasa_Pol_Podst"	M 50.0	BOOL
"M_Bindownica_Poz_Podst"	M 50.1	BOOL
"Auto_Reczny"	M 120.0	BOOL	// auto-1;reczny 0
"Auto_Reczny_3"	M 120.1	BOOL
"PB_Stop_Panel"	M 120.3	BOOL
"Test_Lamp"	M 121.0	BOOL
"Help_Lam_Czerwona"	M 122.0	BOOL
"Help_Lam_Strzal_Tas"	M 122.1	BOOL
"Help_Lam_pb_strefa"	M 122.2	BOOL
"Help_Lam_pb_reczny"	M 122.3	BOOL
"Help_Lam_pb_auto"	M 122.4	BOOL
"Help_Lam_pb_reset"	M 122.5	BOOL
"Help_lam_pb_stop"	M 122.6	BOOL
"Help_Lam_pb_start"	M 122.7	BOOL
"Help_Lam_Biala"	M 123.1	BOOL
"Help_Lam_Blad_Lini"	M 123.2	BOOL
"Help_Lamp_Zielona"	M 123.3	BOOL
"Help_M182.2"	M 180.2	BOOL
"Help_M180.3"	M 180.3	BOOL
"Komunikacja_OK"	M 181.0	BOOL
"M_Miganie_200ms"	M 200.0	BOOL
"M_Miganie_500ms"	M 200.1	BOOL
"M_Miganie_100ms"	M 200.2	BOOL
"BA_Bindownica_Nie_Podst"	M 210.0	BOOL
"Bindownica_Brak_Bezp"	M 210.1	BOOL
"Blad_Foto_Tasma_1"	M 210.2	BOOL
"Blad_Foro_Tasma_2"	M 210.3	BOOL
"Blad_Foto_Tasma_4"	M 210.4	BOOL
"M_Binownica_Blad"	M 210.5	BOOL
"Blad_Fotokomorek_Obr"	M 210.6	BOOL
"Obr_Nie_W_Pozycji"	M 210.7	BOOL
"Byte_Bledu"	MB 10	BYTE
"Nowe_Slowo"	MD 20	DWORD
"Stare_Slowo"	MD 24	DWORD
"Nowe_Slowo_1"	MD 400	DWORD
"Stare_Slowo_1"	MD 404	DWORD
"Nowe_Slowo_2"	MD 408	DWORD
"Stare_Slowo_2"	MD 412	DWORD
"Nowe_Slowo_do_Freeze"	MD 416	DWORD
"Stare_Slowo_do_Freeze"	MD 420	DWORD
"Help_MW12"	MW 12	WORD
"Help_MW14"	MW 14	INT
"Help_MW16"	MW 16	S5TIME
"Help_MW_30"	MW 30	INT
"I/O_FLT1"	OB 82	OB 82	// I/O Point Fault 1
"RACK_FLT"	OB 86	OB 86	// Loss of Rack Fault
"COMPLETE RESTART"	OB 100	OB 100	// Complete Restart
"PROG_ERR"	OB 121	OB 121	// Programming Error
"Lampka_Blad_Bind"	Q 0.0	BOOL
"Lampka_Strzal_Tasmy"	Q 0.1	BOOL
"Lampka_pb_Strefa_Bezp"	Q 0.2	BOOL
"Lampka_pb_Reczny"	Q 0.3	BOOL
"Lampka_pb_Auto"	Q 0.4	BOOL
"Lampka_pb_Reset"	Q 0.5	BOOL
"Lampka_pb_Stop"	Q 0.6	BOOL
"Lampka_pb_Cykl_Start"	Q 0.7	BOOL
"Zawor_Prasa"	Q 1.0	BOOL
"Zezw_na_prace_Bind"	Q 1.1	BOOL
"o_Start_Wiazania"	Q 1.2	BOOL
"rez_q_1_3"	Q 1.3	BOOL
"rez_q_1_4"	Q 1.4	BOOL
"rez_q_1_5"	Q 1.5	BOOL
"Lampka_Lewo_Ok"	Q 1.6	BOOL
"Lampka_Prawo_Ok"	Q 1.7	BOOL
"Reset_P_Bezp"	Q 8.0	BOOL
"Lampka_Biala"	Q 8.1	BOOL
"Lampka_Blad_Lini"	Q 8.2	BOOL
"Lampa_Zielona"	Q 8.3	BOOL
"Silownik_Etykiet"	Q 8.4	BOOL
"Drukuj_Etykiete"	Q 8.5	BOOL
"Zalacz_Skaner"	Q 8.6	BOOL
"Rezerwa_Q_4_7"	Q 8.7	BOOL
"Lampka_Obraz_W_Pamieci"	Q 9.0	BOOL
"Reset_P_Bepz_Strefa"	Q 9.1	BOOL
"TON"	SFB 4	SFB 4	// Generate an On Delay
"READ_CLK"	SFC 1	SFC 1	// Read System Clock
"WR_REC"	SFC 58	SFC 58	// Write Data Record
"RD_REC"	SFC 59	SFC 59	// Read a Data Record
"Auto_Ghost_Mode"	T 37	TIMER
"SEW_Model"	UDT 1	UDT 1	// Model SEW'a
"CROSS_Model"	UDT 2	UDT 2
"ESTOP_Model"	UDT 3	UDT 3
"BRAMA_Model"	UDT 4	UDT 4
"PB_Model"	UDT 5	UDT 5	// Model przycisku
"OBROTOWA_Model"	UDT 6	UDT 6	// Model sygnalow z bandy obrotowej
"CZUJNIKI_1_Model"	UDT 7	UDT 7	// Model czujnikow na obrotnicy
"CZUJNIKI_2_Model"	UDT 8	UDT 8
"S_Model"	UDT 9	UDT 9
"CZUJNIKI_3_MODEL"	UDT 10	UDT 10
"OBROTOWA_2_MODEL"	UDT 11	UDT 11
"RESET_MODEL"	UDT 12	UDT 12
"Wzor_Pracy"	UDT 20	UDT 20
"VAT_1"	VAT 1	
"VAT_Para"	VAT 5	
END_SYMBOL_TABLE

TYPE "SEW_Model"	// UDT 1
VERSION : 0.1
  STRUCT
   Silnik_OK : BOOL ;	//Silnik ok
   Rezerwa_Silnik : BOOL ;
   Foto_1 : BOOL ;	//Wejscie SEW 1
   Foto_2 : BOOL ;	//Wejscie SEW 2
   C_Wise : BOOL ;	//ClockWise
   CC_Wise : BOOL ;	//CounterClockWise
   Wolno : BOOL ;	//Wolno
   S_Bit : BOOL ;	//Bit bezpieczenstwa
   Zez_Do_Pop : BOOL ;	//Zezwolenie do poprzedniej
   Paleta_Dost_do_Pop : BOOL ;	//Potwierdzenie dostarczenia
   Zabierz_do_Nast : BOOL ;	//Przejecie palety do nast
   Paleta_Poprawna : BOOL ;	//Wykorzystywane do monitoringu
   Res_1_4 : BOOL ;
   Res_1_5 : BOOL ;
   Zez_Reczny_do_Pop : BOOL ;	//Zezwolenie na reczny tyl
   Zez_Reczny_do_Nast : BOOL ;	//Zezwolenie na reczny przod
  END_STRUCT ;	
END_TYPE

TYPE "CROSS_Model"	// UDT 2
VERSION : 0.1
  STRUCT
   OSSD_Tor_1_1 : BOOL ;
   OSSD_Tor_1_2 : BOOL ;
   OSSD_Tor_2_1 : BOOL ;
   OSSD_Tor_2_2 : BOOL ;
   Rez_0_4 : BOOL ;
   Rez_0_5 : BOOL ;
   Rez_0_6 : BOOL ;
   Rez_0_7 : BOOL ;
   Rez_1_0 : BOOL ;
   Rez_1_1 : BOOL ;
   Rez_1_2 : BOOL ;
   Rez_1_3 : BOOL ;
   Rez_1_4 : BOOL ;
   Rez_1_5 : BOOL ;
   Rez_1_6 : BOOL ;
   Rez_1_7 : BOOL ;
  END_STRUCT ;	
END_TYPE

TYPE "ESTOP_Model"	// UDT 3
VERSION : 0.1
  STRUCT
   EStop_Tor_1_1 : BOOL ;
   EStop_Tor_1_2 : BOOL ;
   EStop_Tor_2_1 : BOOL ;
   EStop_Tor_2_2 : BOOL ;
   Rez_0_4 : BOOL ;
   Rez_0_5 : BOOL ;
   Rez_0_6 : BOOL ;
   Rez_0_7 : BOOL ;
   Rez_1_0 : BOOL ;
   Rez_1_1 : BOOL ;
   Rez_1_2 : BOOL ;
   Rez_1_3 : BOOL ;
   Rez_1_4 : BOOL ;
   Rez_1_5 : BOOL ;
   Rez_1_6 : BOOL ;
   Rez_1_7 : BOOL ;
  END_STRUCT ;	
END_TYPE

TYPE "PB_Model"	// UDT 5
VERSION : 0.1
  STRUCT
   Przycisk_Start : BOOL ;	//Start i reset ob. bezp
   Czujnik_Kolizji : BOOL ;
   Rez_0_2 : BOOL ;
   Rez_0_3 : BOOL ;
   Rez_0_4 : BOOL ;
   Rez_0_5 : BOOL ;
   Rez_0_6 : BOOL ;
   Rez_0_7 : BOOL ;
   Rez_1_0 : BOOL ;
   Rez_1_1 : BOOL ;
   Rez_1_2 : BOOL ;
   Rez_1_3 : BOOL ;
   Rez_1_4 : BOOL ;
   Rez_1_5 : BOOL ;
   Rez_1_6 : BOOL ;
   Rez_1_7 : BOOL ;
  END_STRUCT ;	
END_TYPE

TYPE "OBROTOWA_Model"	// UDT 6
VERSION : 0.1
  STRUCT
   Silnik_OK : BOOL ;	//Silnik ok
   Rezerwa_Silnik : BOOL ;
   Foto_1 : BOOL ;	//Wejscie SEW 1
   Foto_2 : BOOL ;	//Wejscie SEW 2
   C_Wise : BOOL ;	//ClockWise
   CC_Wise : BOOL ;	//CounterClockWise
   Wolno : BOOL ;	//Wolno
   S_Bit : BOOL ;	//Bit bezpieczenstwa
   Zez_Do_Pop_Wlot_1 : BOOL ;	//Zezwolenie do poprzedniej
   Potw_Dost_Wlot_1 : BOOL ;	//Potwierdzenie dostarczenia
   Zez_Do_Pop_Wlot_2 : BOOL ;	//Wykorzystywane do monitoringu
   Potw_Dost_Wlot_2 : BOOL ;
   Przejmij_Palete : BOOL ;	//Przejecie palety do nast
   Rez_1_6 : BOOL ;
   Paleta_Poprawna_1 : BOOL ;	//Wykorzystywane do monitoringu
  END_STRUCT ;	
END_TYPE

TYPE "CZUJNIKI_1_Model"	// UDT 7
VERSION : 0.1
  STRUCT
   Czujnik_0_St : BOOL ;
   Czujnik_Ham_0_St : BOOL ;
   Czujnik_Ham_90_St : BOOL ;
   Czujnik_90_St : BOOL ;
   Rez_0_4 : BOOL ;
   Rez_0_5 : BOOL ;
   Rez_0_6 : BOOL ;
   Rez_0_7 : BOOL ;
   Rez_1_0 : BOOL ;
   Rez_1_1 : BOOL ;
   Rez_1_2 : BOOL ;
   Rez_1_3 : BOOL ;
   Rez_1_4 : BOOL ;
   Rez_1_5 : BOOL ;
   Rez_1_6 : BOOL ;
   Rez_1_7 : BOOL ;
  END_STRUCT ;	
END_TYPE

TYPE "CZUJNIKI_2_Model"	// UDT 8
VERSION : 0.1
  STRUCT
   Czujnik_45_St_CW : BOOL ;
   Czujnik_45_St_CCW : BOOL ;
   Rez_0_2 : BOOL ;
   Rez_0_3 : BOOL ;
   Rez_0_4 : BOOL ;
   Rez_0_5 : BOOL ;
   Rez_0_6 : BOOL ;
   Rez_0_7 : BOOL ;
   Rez_1_0 : BOOL ;
   Rez_1_1 : BOOL ;
   Rez_1_2 : BOOL ;
   Rez_1_3 : BOOL ;
   Rez_1_4 : BOOL ;
   Rez_1_5 : BOOL ;
   Rez_1_6 : BOOL ;
   Rez_1_7 : BOOL ;
  END_STRUCT ;	
END_TYPE

TYPE "S_Model"	// UDT 9
VERSION : 0.1
  STRUCT
   Silnik_OK : BOOL ;	//Silnik ok
   Rezerwa_Silnik : BOOL ;
   Foto_1 : BOOL ;	//Wejscie SEW 1
   Foto_2 : BOOL ;	//Wejscie SEW 2
   C_Wise : BOOL ;	//ClockWise
   CC_Wise : BOOL ;	//CounterClockWise
   Wolno : BOOL ;	//Wolno
   S_Bit : BOOL ;	//Bit bezpieczenstwa
   Zez_Do_Pop_Wlot_1 : BOOL ;	//Zezwolenie do poprzedniej
   Potw_Dost_Wlot_1 : BOOL ;	//Potwierdzenie dostarczenia
   Zez_Do_Pop_Wlot_2 : BOOL ;	//Wykorzystywane do monitoringu
   Potw_Dost_Wlot_2 : BOOL ;
   Przejmij_Palete : BOOL ;	//Przejecie palety do nast
   Rez_1_6 : BOOL ;
   Paleta_Poprawna_1 : BOOL ;	//Wykorzystywane do monitoringu
  END_STRUCT ;	
END_TYPE

TYPE "CZUJNIKI_3_MODEL"	// UDT 10
VERSION : 0.1
  STRUCT
   Czujnik_Ham_180_St : BOOL ;
   Czujnik_180_St : BOOL ;
   Czujnik_Ham_270_St : BOOL ;
   Czujnik_270_St : BOOL ;
   Rez_0_4 : BOOL ;
   Rez_0_5 : BOOL ;
   Rez_0_6 : BOOL ;
   Rez_0_7 : BOOL ;
   Rez_1_0 : BOOL ;
   Rez_1_1 : BOOL ;
   Rez_1_2 : BOOL ;
   Rez_1_3 : BOOL ;
   Rez_1_4 : BOOL ;
   Rez_1_5 : BOOL ;
   Rez_1_6 : BOOL ;
   Rez_1_7 : BOOL ;
  END_STRUCT ;	
END_TYPE

TYPE "OBROTOWA_2_MODEL"	// UDT 11
VERSION : 0.1
  STRUCT
   Silnik_OK : BOOL ;	//Silnik ok
   Rezerwa_Silnik : BOOL ;
   Foto_1 : BOOL ;	//Wejscie SEW 1
   Foto_2 : BOOL ;	//Wejscie SEW 2
   C_Wise : BOOL ;	//ClockWise
   CC_Wise : BOOL ;	//CounterClockWise
   Wolno : BOOL ;	//Wolno
   S_Bit : BOOL ;	//Bit bezpieczenstwa
   Res_1_0 : BOOL ;	//Zezwolenie do poprzedniej
   Res_1_1 : BOOL ;	//Potwierdzenie dostarczenia
   Res_1_2 : BOOL ;	//Potwierdzenie dostarczenia
   Res_1_3 : BOOL ;	//Potwierdzenie dostarczenia
   Res_1_4 : BOOL ;	//Potwierdzenie dostarczenia
   Res_1_5 : BOOL ;	//Potwierdzenie dostarczenia
   Res_1_6 : BOOL ;	//Potwierdzenie dostarczenia
   Res_1_7 : BOOL ;	//Potwierdzenie dostarczenia
  END_STRUCT ;	
END_TYPE

TYPE "RESET_MODEL"	// UDT 12
VERSION : 0.1
  STRUCT
   Reset_Wlot : BOOL ;
   Reset_Wylot : BOOL ;
   RES_0_2 : BOOL ;
   RES_0_3 : BOOL ;
   Rez_0_4 : BOOL ;
   Rez_0_5 : BOOL ;
   Rez_0_6 : BOOL ;
   Rez_0_7 : BOOL ;
   Rez_1_0 : BOOL ;
   Rez_1_1 : BOOL ;
   Rez_1_2 : BOOL ;
   Rez_1_3 : BOOL ;
   Rez_1_4 : BOOL ;
   Rez_1_5 : BOOL ;
   Rez_1_6 : BOOL ;
   Rez_1_7 : BOOL ;
  END_STRUCT ;	
END_TYPE

TYPE "Wzor_Pracy"	// UDT 20
VERSION : 0.1
  STRUCT
   wiazanie_poprzeczne : BOOL ;
   wiazanie_wzdluzne : BOOL ;
  END_STRUCT ;	
END_TYPE

FUNCTION_BLOCK "TEST_OBR2"	// FB 2
VERSION : 0.1
VAR
  banda_1 : FB 29;
  banda_2 : FB 29;
  banda_3 : FB 29;
  banda_4 : FB 29;
  banda_11 : FB 30;
  banda_12 : FB 30;
  banda_13 : FB 30;
  banda_14 : FB 30;
  banda_obr_2 : FB 32;
  banda_50 : FB 30;
  banda_51 : FB 30;
  banda_52 : FB 30;
  banda_53 : FB 30;
  banda_54 : FB 30;
  czas_z : FB 21;
  tutu : FB 54;
  poz : FB 58;
END_VAR
VAR_TEMP
  temp_help : TIME ;
END_VAR
BEGIN
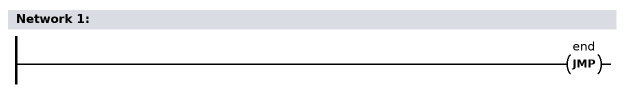
NETWORK
TITLE =
      JU    end;
NETWORK
TITLE =
//Wlot 1
      CALL  #banda_11 (
           S_Marka_Bezpieczenstwa   := "Zawsze_True",
           i_Foto_Koniec            := "pb_Strefa_bezpieczenstwa",
           i_Zez_Od_Nast            := M 102.3,
           i_Paleta_Dost_Od_Nast    := M 102.4,
           Czas_Kontroli_Przejazdu  := T#10S,
           o_Zabierz_Do_Nast        := M 100.0,
           o_Zez_Do_Pop             := M 100.1,
           o_Paleta_Dost_do_Pop     := M 100.2,
           o_Motor_Lewo             := "Lampka_Blad_Bind");
//Wlot 2
      CALL  #banda_12 (
           S_Marka_Bezpieczenstwa   := "Zawsze_True",
           i_Foto_Koniec            := "pb_Reczny",
           i_Zez_Od_Nast            := M 102.1,
           i_Paleta_Dost_Od_Nast    := M 102.2,
           Czas_Kontroli_Przejazdu  := T#10S,
           o_Zabierz_Do_Nast        := M 101.0,
           o_Zez_Do_Pop             := M 101.1,
           o_Paleta_Dost_do_Pop     := M 101.2,
           o_Motor_Lewo             := "Lampka_Strzal_Tasmy");
      CALL  #banda_obr_2 (
           i_Marka_bezpieczenstwa   := "Zawsze_True",
           i_Foto_1                 := "pb_Auto",
           i_Foto_2                 := "pb_Reset",
           i_Zez_od_Nast            := M 103.1,
           i_Zabierz_od_Wlot_1      := M 100.0,
           i_Zabierz_od_Wlot_2      := M 101.0,
           i_Paleta_Odb_Wylot       := M 103.2,
           i_czuj_poz_Wlot_1        := "pb_Tasma_2_Tyl",
           i_czuj_ham_Wlot_1        := "pb_Tasma_2_Przod",
           i_czuj_poz_Wlot_2        := "pb_Tasma_4_Przod",
           i_czuj_ham_Wlot_2        := "pb_Tasma_4_Tyl",
           i_Czuj_poz_45_deg        := "pb_Tasma_3_Tyl",
           i_Czuj_ham_45_deg        := "pb_Tasma_3_Przod",
           i_Foto_Wlot_1            := "pb_Strefa_bezpieczenstwa",
           i_Foto_Wlot_2            := "pb_Reczny",
           i_Etyk_praca_wlacz       := "Bind_Polozenie_Podst",
           i_Etyk_poz_podst         := "Obwod_Bezp_Bindownicy",
           i_Etyk_obraz_w_pamieci   := "Foto_Wozek",
           i_Etyk_syg_gotowosci     := "Start_Koniec_Wiazania",
           i_Etyk_brak_materialu    := "Bindownica_Auto",
           i_Etyk_Przycisk_Drukuj   := "rez_i_2_5",
           o_Zez_do_Wlot_1          := M 102.3,
           o_Zez_do_Wlot_2          := M 102.1,
           o_Paleta_Dost_Wlot_1     := M 102.4,
           o_Paleta_Dost_Wlot_2     := M 102.2,
           o_Zabierz_do_Nast        := M 102.0,
           o_Motor_1_lewo           := "Lampka_pb_Strefa_Bezp",
           o_Motor_1_prawo          := "Lampka_pb_Reczny",
           o_Motor_2_obr_s_Wlot_1   := "Zawor_Prasa",
           o_Motor_2_obr_s_Wlot_2   := "Zezw_na_prace_Bind",
           o_Silownik_etykiety      := "Lampka_Prawo_Ok",
           o_Drukuj_Etykiete        := "Lampka_Lewo_Ok",
           o_Zalaczenie_Skanera     := "rez_q_1_5");
      CALL  #banda_14 (
           S_Marka_Bezpieczenstwa   := "Zawsze_True",
           i_Foto_Koniec            := "pb_Stop",
           i_Zabierz_Od_Pop         := M 102.0,
           Czas_Kontroli_Przejazdu  := T#10S,
           o_Zabierz_Do_Nast        := M 103.0,
           o_Zez_Do_Pop             := M 103.1,
           o_Paleta_Dost_do_Pop     := M 103.2,
           o_Motor_Lewo             := "Lampka_pb_Auto");
      BEU;
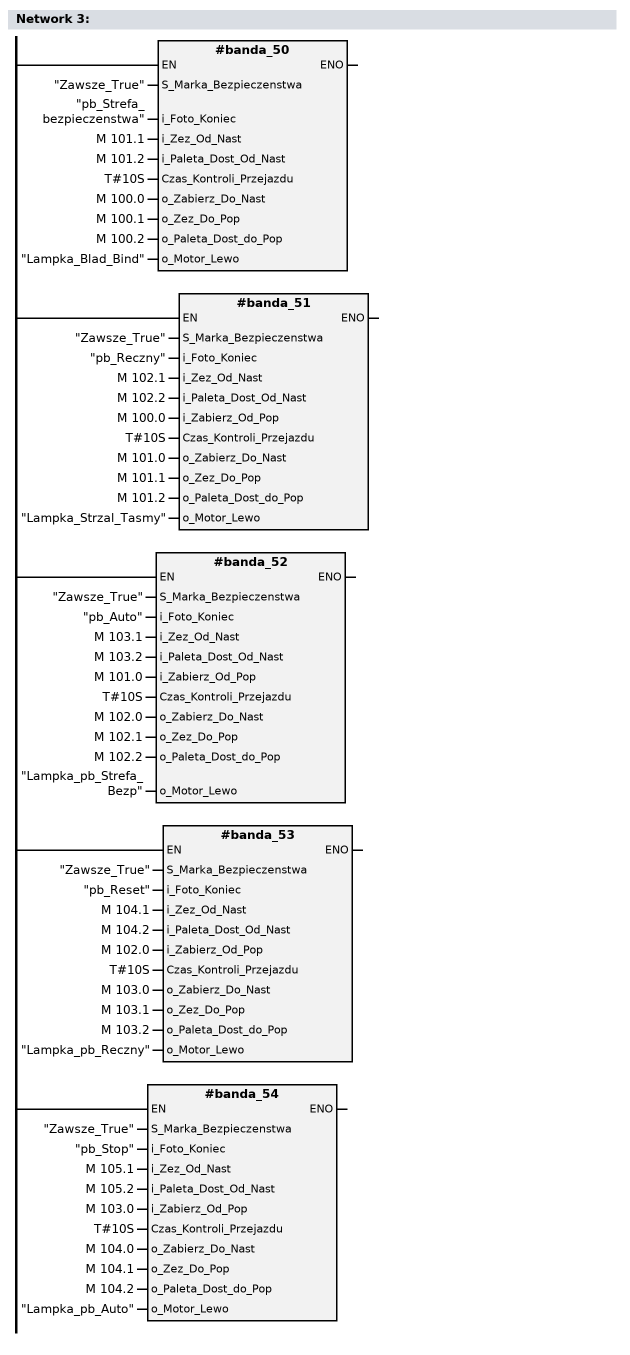
NETWORK
TITLE =
      CALL  #banda_50 (
           S_Marka_Bezpieczenstwa   := "Zawsze_True",
           i_Foto_Koniec            := "pb_Strefa_bezpieczenstwa",
           i_Zez_Od_Nast            := M 101.1,
           i_Paleta_Dost_Od_Nast    := M 101.2,
           Czas_Kontroli_Przejazdu  := T#10S,
           o_Zabierz_Do_Nast        := M 100.0,
           o_Zez_Do_Pop             := M 100.1,
           o_Paleta_Dost_do_Pop     := M 100.2,
           o_Motor_Lewo             := "Lampka_Blad_Bind");
      CALL  #banda_51 (
           S_Marka_Bezpieczenstwa   := "Zawsze_True",
           i_Foto_Koniec            := "pb_Reczny",
           i_Zez_Od_Nast            := M 102.1,
           i_Paleta_Dost_Od_Nast    := M 102.2,
           i_Zabierz_Od_Pop         := M 100.0,
           Czas_Kontroli_Przejazdu  := T#10S,
           o_Zabierz_Do_Nast        := M 101.0,
           o_Zez_Do_Pop             := M 101.1,
           o_Paleta_Dost_do_Pop     := M 101.2,
           o_Motor_Lewo             := "Lampka_Strzal_Tasmy");
      CALL  #banda_52 (
           S_Marka_Bezpieczenstwa   := "Zawsze_True",
           i_Foto_Koniec            := "pb_Auto",
           i_Zez_Od_Nast            := M 103.1,
           i_Paleta_Dost_Od_Nast    := M 103.2,
           i_Zabierz_Od_Pop         := M 101.0,
           Czas_Kontroli_Przejazdu  := T#10S,
           o_Zabierz_Do_Nast        := M 102.0,
           o_Zez_Do_Pop             := M 102.1,
           o_Paleta_Dost_do_Pop     := M 102.2,
           o_Motor_Lewo             := "Lampka_pb_Strefa_Bezp");
      CALL  #banda_53 (
           S_Marka_Bezpieczenstwa   := "Zawsze_True",
           i_Foto_Koniec            := "pb_Reset",
           i_Zez_Od_Nast            := M 104.1,
           i_Paleta_Dost_Od_Nast    := M 104.2,
           i_Zabierz_Od_Pop         := M 102.0,
           Czas_Kontroli_Przejazdu  := T#10S,
           o_Zabierz_Do_Nast        := M 103.0,
           o_Zez_Do_Pop             := M 103.1,
           o_Paleta_Dost_do_Pop     := M 103.2,
           o_Motor_Lewo             := "Lampka_pb_Reczny");
      CALL  #banda_54 (
           S_Marka_Bezpieczenstwa   := "Zawsze_True",
           i_Foto_Koniec            := "pb_Stop",
           i_Zez_Od_Nast            := M 105.1,
           i_Paleta_Dost_Od_Nast    := M 105.2,
           i_Zabierz_Od_Pop         := M 103.0,
           Czas_Kontroli_Przejazdu  := T#10S,
           o_Zabierz_Do_Nast        := M 104.0,
           o_Zez_Do_Pop             := M 104.1,
           o_Paleta_Dost_do_Pop     := M 104.2,
           o_Motor_Lewo             := "Lampka_pb_Auto");
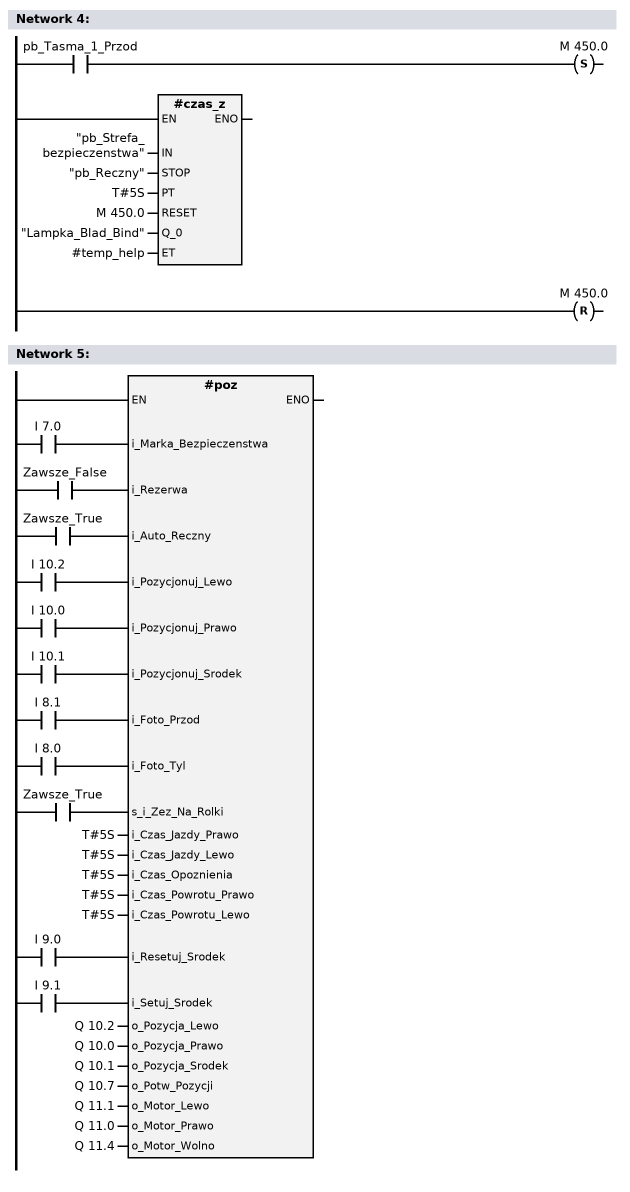
NETWORK
TITLE =
//test nowego timmera 
//
      NOP   0;
      A     "pb_Tasma_1_Przod";
      S     M 450.0;
      CALL  #czas_z (
           IN                       := "pb_Strefa_bezpieczenstwa",
           STOP                     := "pb_Reczny",
           PT                       := T#5S,
           RESET                    := M 450.0,
           Q_0                      := "Lampka_Blad_Bind",
           ET                       := #temp_help);
      SET;
      R     M 450.0;
end:  NOP   0;
NETWORK
TITLE =
      A     I 7.0;
      =     L 4.0;
      BLD   103;
      A     "Zawsze_False";
      =     L 4.1;
      BLD   103;
      A     "Zawsze_True";
      =     L 4.2;
      BLD   103;
      A     I 10.2;
      =     L 4.3;
      BLD   103;
      A     I 10.0;
      =     L 4.4;
      BLD   103;
      A     I 10.1;
      =     L 4.5;
      BLD   103;
      A     I 8.1;
      =     L 4.6;
      BLD   103;
      A     I 8.0;
      =     L 4.7;
      BLD   103;
      A     "Zawsze_True";
      =     L 5.0;
      BLD   103;
      A     I 9.0;
      =     L 5.2;
      BLD   103;
      A     I 9.1;
      =     L 5.3;
      BLD   103;
      CALL  #poz (
           i_Marka_Bezpieczenstwa   := L 4.0,
           i_Rezerwa                := L 4.1,
           i_Auto_Reczny            := L 4.2,
           i_Pozycjonuj_Lewo        := L 4.3,
           i_Pozycjonuj_Prawo       := L 4.4,
           i_Pozycjonuj_Srodek      := L 4.5,
           i_Foto_Przod             := L 4.6,
           i_Foto_Tyl               := L 4.7,
           s_i_Zez_Na_Rolki         := L 5.0,
           i_Czas_Jazdy_Prawo       := T#5S,
           i_Czas_Jazdy_Lewo        := T#5S,
           i_Czas_Opoznienia        := T#5S,
           i_Czas_Powrotu_Prawo     := T#5S,
           i_Czas_Powrotu_Lewo      := T#5S,
           i_Resetuj_Srodek         := L 5.2,
           i_Setuj_Srodek           := L 5.3,
           o_Pozycja_Lewo           := Q 10.2,
           o_Pozycja_Prawo          := Q 10.0,
           o_Pozycja_Srodek         := Q 10.1,
           o_Potw_Pozycji           := Q 10.7,
           o_Motor_Lewo             := Q 11.1,
           o_Motor_Prawo            := Q 11.0,
           o_Motor_Wolno            := Q 11.4);
      NOP   0;
END_FUNCTION_BLOCK

FUNCTION_BLOCK "Czesc_Bindujaca"	// FB 3
//Funkcja odpowiada za sterowanie lini bindujacej
//Uwzgledniony zostal tryb reczny
//
VERSION : 0.1
VAR
  Tasma_1 : FB 33;	//Adres 23
  Tasma_2 : FB 33;	//Adres 24
  Tasma_Obr_3 : FB 34;	//Adres 1 i 15
  Tasma_4 : FB 33;	//Adres 2
  Bin_IN_OUT : FB 57;
  Bind_Obwod_Ok : BOOL ;
  Bind_Poz_Podst : BOOL ;
  Bind_Sygn_Got : BOOL ;
  Bind_Blad : BOOL ;
  Bind_Start_Kon : BOOL ;
  Zaj_Nieb_2 : BOOL ;
  Zaj_Nieb_4 : BOOL ;
  Tasma_Rezerwa_1 : FB 33;
  Tasma_Rezerwa_2 : FB 33;
END_VAR
VAR_TEMP
  Temp_Bit_1 : BOOL ;
END_VAR
BEGIN
NETWORK
TITLE =
//Ten network celowo jest wolny
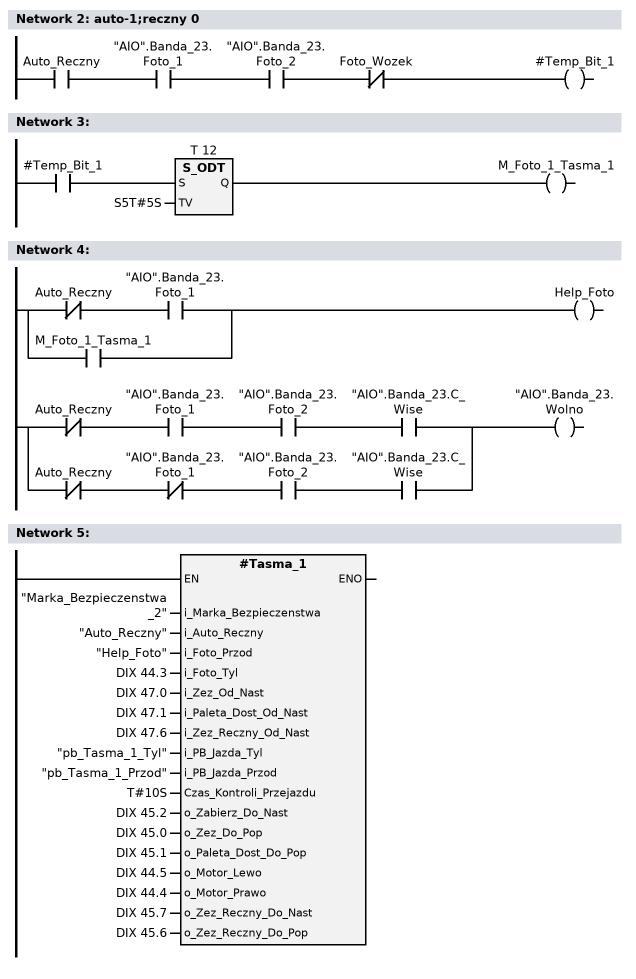
NETWORK
TITLE = auto-1;reczny 0
      A     "Auto_Reczny";
      A     "AIO".Banda_23.Foto_1;
      A     "AIO".Banda_23.Foto_2;
      AN    "Foto_Wozek";
      =     #Temp_Bit_1;
NETWORK
TITLE =
//Opoznienie startu po polozeniu palety
//
      A     #Temp_Bit_1;
      L     S5T#5S;
      SD    T 12;
      NOP   0;
      NOP   0;
      NOP   0;
      A     T 12;
      =     "M_Foto_1_Tasma_1";
NETWORK
TITLE =
//Opoznienie wlotu bandy 1
      AN    "Auto_Reczny";
      A     "AIO".Banda_23.Foto_1;
      O;
      A     "M_Foto_1_Tasma_1";
      =     "Help_Foto";
//Silnik wolno  aby nie spadl z bandy
      AN    "Auto_Reczny";
      A     "AIO".Banda_23.Foto_1;
      A     "AIO".Banda_23.Foto_2;
      A     "AIO".Banda_23.C_Wise;
//      A     "Zawsze_False"
      O;
      AN    "Auto_Reczny";
      AN    "AIO".Banda_23.Foto_1;
      A     "AIO".Banda_23.Foto_2;
      A     "AIO".Banda_23.C_Wise;
      =     "AIO".Banda_23.Wolno;
NETWORK
TITLE =
//Tasma 1 adres 23
      CALL  #Tasma_1 (
           i_Marka_Bezpieczenstwa   := "Marka_Bezpieczenstwa_2",
           i_Auto_Reczny            := "Auto_Reczny",
           i_Foto_Przod             := "Help_Foto",
           i_Foto_Tyl               := DIX 44.3,
           i_Zez_Od_Nast            := DIX 47.0,
           i_Paleta_Dost_Od_Nast    := DIX 47.1,
           i_Zez_Reczny_Od_Nast     := DIX 47.6,
           i_PB_Jazda_Tyl           := "pb_Tasma_1_Tyl",
           i_PB_Jazda_Przod         := "pb_Tasma_1_Przod",
           Czas_Kontroli_Przejazdu  := T#10S,
           o_Zabierz_Do_Nast        := DIX 45.2,
           o_Zez_Do_Pop             := DIX 45.0,
           o_Paleta_Dost_Do_Pop     := DIX 45.1,
           o_Motor_Lewo             := DIX 44.5,
           o_Motor_Prawo            := DIX 44.4,
           o_Zez_Reczny_Do_Nast     := DIX 45.7,
           o_Zez_Reczny_Do_Pop      := DIX 45.6);	//kierunek normalny lini
      NOP   0;
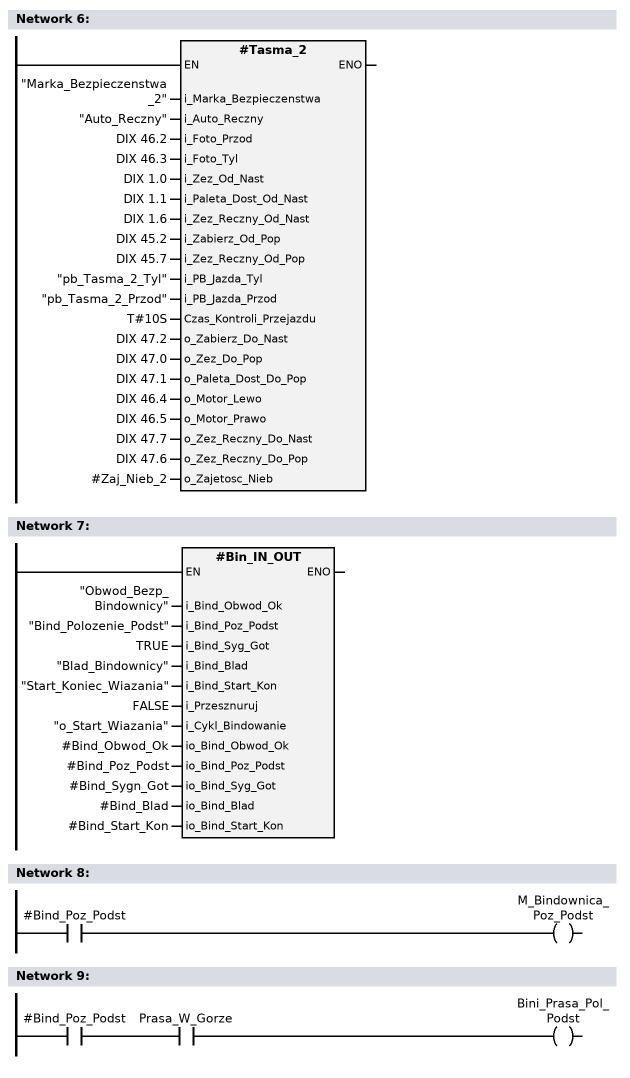
NETWORK
TITLE =
//Tasma 2 adres 24
      CALL  #Tasma_2 (
           i_Marka_Bezpieczenstwa   := "Marka_Bezpieczenstwa_2",
           i_Auto_Reczny            := "Auto_Reczny",
           i_Foto_Przod             := DIX 46.2,
           i_Foto_Tyl               := DIX 46.3,
           i_Zez_Od_Nast            := DIX 1.0,
           i_Paleta_Dost_Od_Nast    := DIX 1.1,
           i_Zez_Reczny_Od_Nast     := DIX 1.6,
           i_Zabierz_Od_Pop         := DIX 45.2,
           i_Zez_Reczny_Od_Pop      := DIX 45.7,
           i_PB_Jazda_Tyl           := "pb_Tasma_2_Tyl",
           i_PB_Jazda_Przod         := "pb_Tasma_2_Przod",
           Czas_Kontroli_Przejazdu  := T#10S,
           o_Zabierz_Do_Nast        := DIX 47.2,
           o_Zez_Do_Pop             := DIX 47.0,
           o_Paleta_Dost_Do_Pop     := DIX 47.1,
           o_Motor_Lewo             := DIX 46.4,
           o_Motor_Prawo            := DIX 46.5,
           o_Zez_Reczny_Do_Nast     := DIX 47.7,
           o_Zez_Reczny_Do_Pop      := DIX 47.6,
           o_Zajetosc_Nieb          := #Zaj_Nieb_2);	//kierunek normalny lini
      NOP   0;
NETWORK
TITLE =
//blok przejsciowy  do bindownicy
//(maskuje sygnal wejscia i wyjscia)
      CALL  #Bin_IN_OUT (
           i_Bind_Obwod_Ok          := "Obwod_Bezp_Bindownicy",
           i_Bind_Poz_Podst         := "Bind_Polozenie_Podst",
           i_Bind_Syg_Got           := TRUE,
           i_Bind_Blad              := "Blad_Bindownicy",
           i_Bind_Start_Kon         := "Start_Koniec_Wiazania",
           i_Przesznuruj            := FALSE,
           i_Cykl_Bindowanie        := "o_Start_Wiazania",
           io_Bind_Obwod_Ok         := #Bind_Obwod_Ok,
           io_Bind_Poz_Podst        := #Bind_Poz_Podst,
           io_Bind_Syg_Got          := #Bind_Sygn_Got,
           io_Bind_Blad             := #Bind_Blad,
           io_Bind_Start_Kon        := #Bind_Start_Kon);
NETWORK
TITLE =
      A     #Bind_Poz_Podst;
      =     "M_Bindownica_Poz_Podst";
NETWORK
TITLE =
      A     #Bind_Poz_Podst;
      A     "Prasa_W_Gorze";
      =     "Bini_Prasa_Pol_Podst";
NETWORK
TITLE =
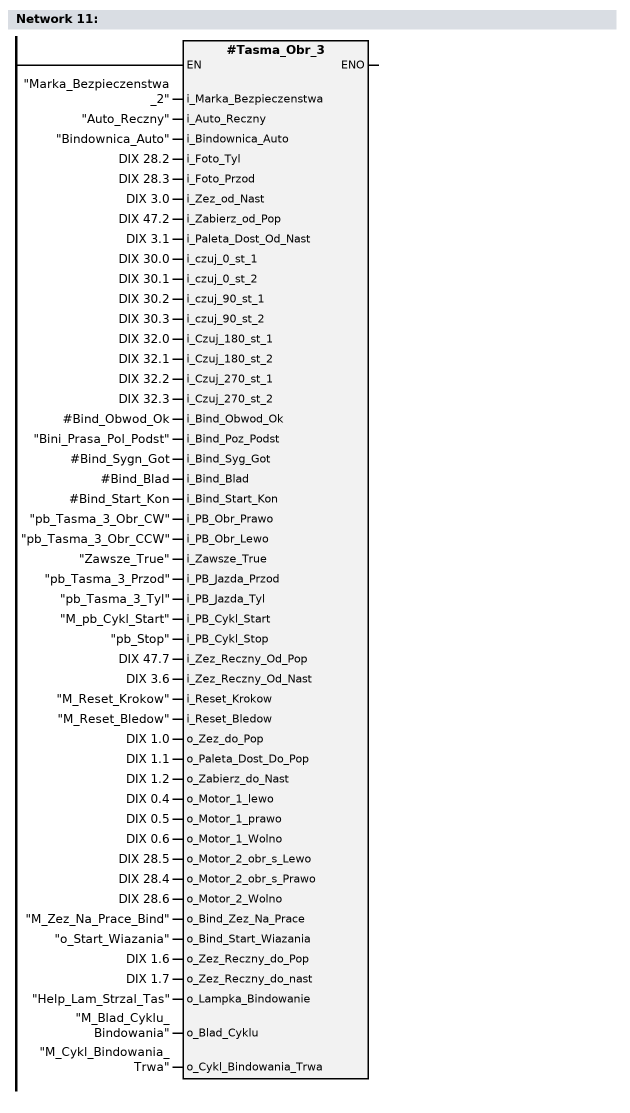
NETWORK
TITLE =
//bindownica z obrotnica
      CALL  #Tasma_Obr_3 (
           i_Marka_Bezpieczenstwa   := "Marka_Bezpieczenstwa_2",
           i_Auto_Reczny            := "Auto_Reczny",
           i_Bindownica_Auto        := "Bindownica_Auto",
           i_Foto_Tyl               := DIX 28.2,
           i_Foto_Przod             := DIX 28.3,
           i_Zez_od_Nast            := DIX 3.0,
           i_Zabierz_od_Pop         := DIX 47.2,
           i_Paleta_Dost_Od_Nast    := DIX 3.1,
           i_czuj_0_st_1            := DIX 30.0,
           i_czuj_0_st_2            := DIX 30.1,
           i_czuj_90_st_1           := DIX 30.2,
           i_czuj_90_st_2           := DIX 30.3,
           i_Czuj_180_st_1          := DIX 32.0,
           i_Czuj_180_st_2          := DIX 32.1,
           i_Czuj_270_st_1          := DIX 32.2,
           i_Czuj_270_st_2          := DIX 32.3,
           i_Bind_Obwod_Ok          := #Bind_Obwod_Ok,
           i_Bind_Poz_Podst         := "Bini_Prasa_Pol_Podst",
           i_Bind_Syg_Got           := #Bind_Sygn_Got,
           i_Bind_Blad              := #Bind_Blad,
           i_Bind_Start_Kon         := #Bind_Start_Kon,
           i_PB_Obr_Prawo           := "pb_Tasma_3_Obr_CW",
           i_PB_Obr_Lewo            := "pb_Tasma_3_Obr_CCW",
           i_Zawsze_True            := "Zawsze_True",
           i_PB_Jazda_Przod         := "pb_Tasma_3_Przod",
           i_PB_Jazda_Tyl           := "pb_Tasma_3_Tyl",
           i_PB_Cykl_Start          := "M_pb_Cykl_Start",
           i_PB_Cykl_Stop           := "pb_Stop",
           i_Zez_Reczny_Od_Pop      := DIX 47.7,
           i_Zez_Reczny_Od_Nast     := DIX 3.6,
           i_Reset_Krokow           := "M_Reset_Krokow",
           i_Reset_Bledow           := "M_Reset_Bledow",
           o_Zez_do_Pop             := DIX 1.0,
           o_Paleta_Dost_Do_Pop     := DIX 1.1,
           o_Zabierz_do_Nast        := DIX 1.2,
           o_Motor_1_lewo           := DIX 0.4,
           o_Motor_1_prawo          := DIX 0.5,
           o_Motor_1_Wolno          := DIX 0.6,
           o_Motor_2_obr_s_Lewo     := DIX 28.5,
           o_Motor_2_obr_s_Prawo    := DIX 28.4,
           o_Motor_2_Wolno          := DIX 28.6,
           o_Bind_Zez_Na_Prace      := "M_Zez_Na_Prace_Bind",
           o_Bind_Start_Wiazania    := "o_Start_Wiazania",
           o_Zez_Reczny_do_Pop      := DIX 1.6,
           o_Zez_Reczny_do_nast     := DIX 1.7,
           o_Lampka_Bindowanie      := "Help_Lam_Strzal_Tas",
           o_Blad_Cyklu             := "M_Blad_Cyklu_Bindowania",
           o_Cykl_Bindowania_Trwa   := "M_Cykl_Bindowania_Trwa");
NETWORK
TITLE = Zezwolenie na prase reczny
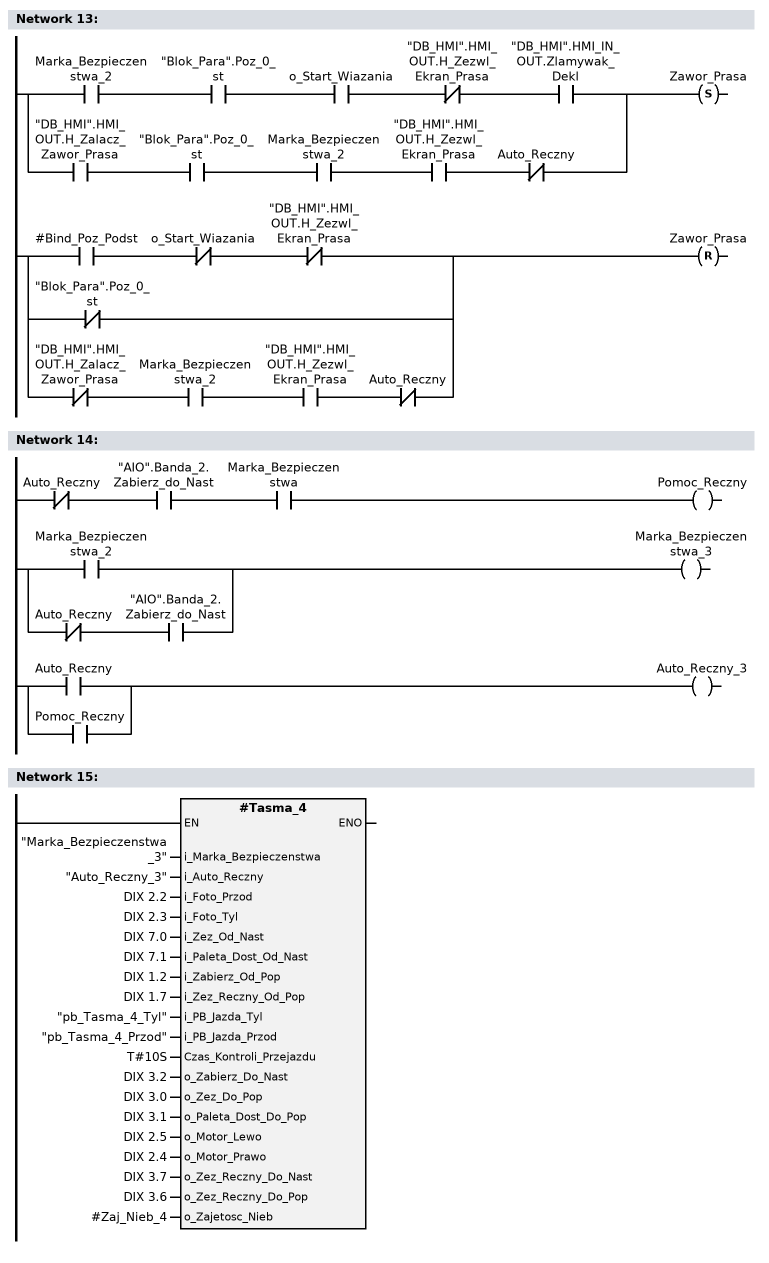
NETWORK
TITLE =
      A(;
      A     "Marka_Bezpieczenstwa_2";
      A     "Blok_Para".Poz_0_st;
      A     "o_Start_Wiazania";
      AN    "DB_HMI".HMI_OUT.H_Zezwl_Ekran_Prasa;
      A     "DB_HMI".HMI_IN_OUT.Zlamywak_Dekl;
      O;
      A     "DB_HMI".HMI_OUT.H_Zalacz_Zawor_Prasa;
      A     "Blok_Para".Poz_0_st;
      A     "Marka_Bezpieczenstwa_2";
      A     "DB_HMI".HMI_OUT.H_Zezwl_Ekran_Prasa;
      AN    "Auto_Reczny";
      );
      S     "Zawor_Prasa";
      A(;
      A     #Bind_Poz_Podst;
      AN    "o_Start_Wiazania";
      AN    "DB_HMI".HMI_OUT.H_Zezwl_Ekran_Prasa;
      ON    "Blok_Para".Poz_0_st;
      O;
      AN    "DB_HMI".HMI_OUT.H_Zalacz_Zawor_Prasa;
      A     "Marka_Bezpieczenstwa_2";
      A     "DB_HMI".HMI_OUT.H_Zezwl_Ekran_Prasa;
      AN    "Auto_Reczny";
      );
      R     "Zawor_Prasa";
      NOP   0;
NETWORK
TITLE =
//Nowa Marka bepieczenstwa na wyjazd
//Marka bepieczenstwa przejsciowa
      AN    "Auto_Reczny";
      A     "AIO".Banda_2.Zabierz_do_Nast;
      A     "Marka_Bezpieczenstwa";
      =     "Pomoc_Reczny";
      A     "Marka_Bezpieczenstwa_2";
      O;
      AN    "Auto_Reczny";
      A     "AIO".Banda_2.Zabierz_do_Nast;
      =     "Marka_Bezpieczenstwa_3";
//Jezeli marka bezpieczenstwa 3 auto zalaczone
      A     "Auto_Reczny";
      O;
      A     "Pomoc_Reczny";
      =     "Auto_Reczny_3";
NETWORK
TITLE =
//Tasma 4 adres 2
//Ta tasma pod wzgledem bezpieczenstwa nalezy do lini i bindownicy
//Nastepna banda jest obrotnica
//
//
//
      CALL  #Tasma_4 (
           i_Marka_Bezpieczenstwa   := "Marka_Bezpieczenstwa_3",
           i_Auto_Reczny            := "Auto_Reczny_3",
           i_Foto_Przod             := DIX 2.2,
           i_Foto_Tyl               := DIX 2.3,
           i_Zez_Od_Nast            := DIX 7.0,
           i_Paleta_Dost_Od_Nast    := DIX 7.1,
           i_Zabierz_Od_Pop         := DIX 1.2,
           i_Zez_Reczny_Od_Pop      := DIX 1.7,
           i_PB_Jazda_Tyl           := "pb_Tasma_4_Tyl",
           i_PB_Jazda_Przod         := "pb_Tasma_4_Przod",
           Czas_Kontroli_Przejazdu  := T#10S,
           o_Zabierz_Do_Nast        := DIX 3.2,
           o_Zez_Do_Pop             := DIX 3.0,
           o_Paleta_Dost_Do_Pop     := DIX 3.1,
           o_Motor_Lewo             := DIX 2.5,
           o_Motor_Prawo            := DIX 2.4,
           o_Zez_Reczny_Do_Nast     := DIX 3.7,
           o_Zez_Reczny_Do_Pop      := DIX 3.6,
           o_Zajetosc_Nieb          := #Zaj_Nieb_4);	//kierunek normalny lini
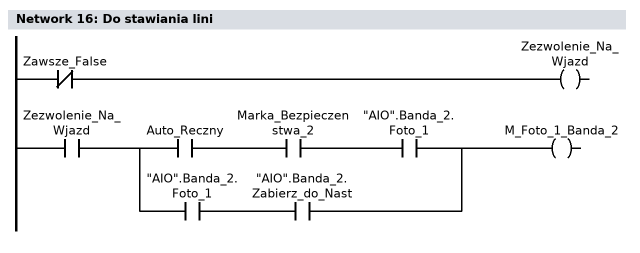
NETWORK
TITLE = Do stawiania lini
//Banda 2. Uznawana za Wlot 1
//Uwaga By dzialolo nalezy wymusic true
      AN    "Zawsze_False";
      =     "Zezwolenie_Na_Wjazd";
//--
      A     "Zezwolenie_Na_Wjazd";
      A(;
      A     "Auto_Reczny";
      A     "Marka_Bezpieczenstwa_2";
      A     "AIO".Banda_2.Foto_1;
      O;
      A     "AIO".Banda_2.Foto_1;
      A     "AIO".Banda_2.Zabierz_do_Nast;
      );
      =     "M_Foto_1_Banda_2";
END_FUNCTION_BLOCK

